LIN {X 0,Y 467.549,Z 626.363,A -85,B 0,C 180,E1 -7509.148,E2 -7509.148} C_VEL
LIN {X 0,Y 467.561,Z 626.367,A -85,B 0,C 180,E1 -7511.405,E2 -7511.405} C_VEL
LIN {X 0,Y 467.569,Z 626.37,A -85,B 0,C 180,E1 -7515.052,E2 -7515.052} C_VEL
LIN {X 0,Y 467.563,Z 626.367,A -85,B 0,C 180,E1 -7518.726,E2 -7518.726} C_VEL
LIN {X 0,Y 467.552,Z 626.355,A -85,B 0,C 180,E1 -7521.954,E2 -7521.954} C_VEL
LIN {X 0,Y 467.559,Z 626.366,A -85,B 0,C 180,E1 -7525.166,E2 -7525.166} C_VEL
LIN {X 0,Y 467.585,Z 626.36,A -85,B 0,C 180,E1 -7528.26,E2 -7528.26} C_VEL
LIN {X 0,Y 467.556,Z 626.368,A -85,B 0,C 180,E1 -7531.249,E2 -7531.249} C_VEL
LIN {X 0,Y 467.579,Z 626.36,A -85,B 0,C 180,E1 -7534.401,E2 -7534.401} C_VEL
LIN {X 0,Y 467.579,Z 626.359,A -85,B 0,C 180,E1 -7536.996,E2 -7536.996} C_VEL
LIN {X 0,Y 467.626,Z 626.359,A -85,B 0,C 180,E1 -7539.777,E2 -7539.777} C_VEL
LIN {X 0,Y 467.601,Z 626.35,A -85,B 0,C 180,E1 -7542.506,E2 -7542.506} C_VEL
LIN {X 0,Y 467.609,Z 626.36,A -85,B 0,C 180,E1 -7545.196,E2 -7545.196} C_VEL
LIN {X 0,Y 467.659,Z 626.352,A -85,B 0,C 180,E1 -7547.854,E2 -7547.854} C_VEL
LIN {X 0,Y 467.673,Z 626.349,A -85,B 0,C 180,E1 -7551.357,E2 -7551.357} C_VEL
LIN {X 0,Y 467.716,Z 626.348,A -85,B 0,C 180,E1 -7553.962,E2 -7553.962} C_VEL
LIN {X 0,Y 467.854,Z 626.329,A -85,B 0,C 180,E1 -7557.417,E2 -7557.417} C_VEL
LIN {X 0,Y 467.885,Z 626.326,A -85,B 0,C 180,E1 -7560,E2 -7560} C_VEL
LIN {X 0,Y 467.861,Z 626.327,A -85,B 0,C 180,E1 -7562.583,E2 -7562.583} C_VEL
LIN {X 0,Y 467.725,Z 626.348,A -85,B 0,C 180,E1 -7566.037,E2 -7566.037} C_VEL
LIN {X 0,Y 467.683,Z 626.349,A -85,B 0,C 180,E1 -7568.643,E2 -7568.643} C_VEL
LIN {X 0,Y 467.659,Z 626.358,A -85,B 0,C 180,E1 -7572.145,E2 -7572.145} C_VEL
LIN {X 0,Y 467.67,Z 626.353,A -85,B 0,C 180,E1 -7575.893,E2 -7575.893} C_VEL
LIN {X 0,Y 467.627,Z 626.353,A -85,B 0,C 180,E1 -7579.307,E2 -7579.307} C_VEL
LIN {X 0,Y 467.537,Z 626.373,A -85,B 0,C 180,E1 -7582.074,E2 -7582.074} C_VEL
LIN {X 0,Y 467.588,Z 626.361,A -85,B 0,C 180,E1 -7584.888,E2 -7584.888} C_VEL
LIN {X 0,Y 467.622,Z 626.356,A -85,B 0,C 180,E1 -7587.769,E2 -7587.769} C_VEL
LIN {X 0,Y 467.57,Z 626.362,A -85,B 0,C 180,E1 -7591.045,E2 -7591.045} C_VEL
LIN {X 0,Y 467.59,Z 626.366,A -85,B 0,C 180,E1 -7594.242,E2 -7594.242} C_VEL
LIN {X 0,Y 467.55,Z 626.366,A -85,B 0,C 180,E1 -7597.186,E2 -7597.186} C_VEL
LIN {X 0,Y 467.597,Z 626.364,A -85,B 0,C 180,E1 -7600.262,E2 -7600.262} C_VEL
LIN {X 0,Y 467.588,Z 626.368,A -85,B 0,C 180,E1 -7602.567,E2 -7602.567} C_VEL
LIN {X 0,Y 467.572,Z 626.364,A -85,B 0,C 180,E1 -7605.053,E2 -7605.053} C_VEL
LIN {X 0,Y 467.59,Z 626.36,A -85,B 0,C 180,E1 -7607.44,E2 -7607.44} C_VEL
LIN {X 0,Y 467.584,Z 626.368,A -85,B 0,C 180,E1 -7610.855,E2 -7610.855} C_VEL
LIN {X 0,Y 467.565,Z 626.368,A -85,B 0,C 180,E1 -7614.26,E2 -7614.26} C_VEL
LIN {X 0,Y 467.584,Z 626.365,A -85,B 0,C 180,E1 -7617.321,E2 -7617.321} C_VEL
LIN {X 0,Y 467.572,Z 626.369,A -85,B 0,C 180,E1 -7620.667,E2 -7620.667} C_VEL
LIN {X 0,Y 467.653,Z 626.484,A -85,B 0,C 180,E1 -7621.654,E2 -7621.654} C_VEL
LIN {X 0,Y 470.749,Z 640.596,A -85,B 0,C 180,E1 -7624.125,E2 -7624.125} C_VEL
LIN {X 0,Y 471.136,Z 644.928,A -85,B 0,C 180,E1 -7624.84,E2 -7624.84} C_VEL
LIN {X 0,Y 469.974,Z 666.892,A -85,B 0,C 180,E1 -7628.277,E2 -7628.277} C_VEL
LIN {X 0,Y 469.639,Z 674.02,A -85,B 0,C 180,E1 -7629.383,E2 -7629.383} C_VEL
LIN {X 0,Y 473.403,Z 695.857,A -85,B 0,C 180,E1 -7629.896,E2 -7629.896} C_VEL
LIN {X 0,Y 472.198,Z 812.498,A -85,B 0,C 180,E1 -7631.702,E2 -7631.702} C_VEL
LIN {X 0,Y 471.755,Z 827.182,A -85,B 0,C 180,E1 -7632.108,E2 -7632.108} C_VEL
LIN {X 0,Y 471.281,Z 840.517,A -85,B 0,C 180,E1 -7632.647,E2 -7632.647} C_VEL
LIN {X 0,Y 470.687,Z 853.287,A -85,B 0,C 180,E1 -7633.329,E2 -7633.329} C_VEL
LIN {X 0,Y 470.047,Z 865.621,A -85,B 0,C 180,E1 -7634.165,E2 -7634.165} C_VEL
LIN {X 0,Y 469.361,Z 877.324,A -85,B 0,C 180,E1 -7635.142,E2 -7635.142} C_VEL
LIN {X 0,Y 468.755,Z 887.065,A -85,B 0,C 180,E1 -7636.12,E2 -7636.12} C_VEL
LIN {X 0,Y 468.168,Z 897.352,A -85,B 0,C 180,E1 -7637.359,E2 -7637.359} C_VEL
LIN {X 0,Y 467.713,Z 906.781,A -85,B 0,C 180,E1 -7638.735,E2 -7638.735} C_VEL
LIN {X 0,Y 467.263,Z 915.33,A -85,B 0,C 180,E1 -7640.258,E2 -7640.258} C_VEL
LIN {X 0,Y 466.964,Z 922.224,A -85,B 0,C 180,E1 -7641.78,E2 -7641.78} C_VEL
LIN {X 0,Y 466.825,Z 926.979,A -85,B 0,C 180,E1 -7643.082,E2 -7643.082} C_VEL
LIN {X 0,Y 466.757,Z 931.907,A -85,B 0,C 180,E1 -7644.817,E2 -7644.817} C_VEL
LIN {X 0,Y 466.681,Z 935.332,A -85,B 0,C 180,E1 -7646.546,E2 -7646.546} C_VEL
LIN {X 0,Y 466.625,Z 937.357,A -85,B 0,C 180,E1 -7648.274,E2 -7648.274} C_VEL
LIN {X 0,Y 466.596,Z 938.027,A -85,B 0,C 180,E1 -7650,E2 -7650} C_VEL
LIN {X 0,Y 466.625,Z 937.354,A -85,B 0,C 180,E1 -7651.726,E2 -7651.726} C_VEL
LIN {X 0,Y 466.681,Z 935.327,A -85,B 0,C 180,E1 -7653.453,E2 -7653.453} C_VEL
LIN {X 0,Y 466.757,Z 931.896,A -85,B 0,C 180,E1 -7655.183,E2 -7655.183} C_VEL
LIN {X 0,Y 466.822,Z 926.957,A -85,B 0,C 180,E1 -7656.917,E2 -7656.917} C_VEL
LIN {X 0,Y 467.051,Z 920.373,A -85,B 0,C 180,E1 -7658.654,E2 -7658.654} C_VEL
LIN {X 0,Y 467.334,Z 913.049,A -85,B 0,C 180,E1 -7660.178,E2 -7660.178} C_VEL
LIN {X 0,Y 467.853,Z 903.988,A -85,B 0,C 180,E1 -7661.7,E2 -7661.7} C_VEL
LIN {X 0,Y 468.348,Z 894.482,A -85,B 0,C 180,E1 -7663.008,E2 -7663.008} C_VEL
LIN {X 0,Y 468.929,Z 883.967,A -85,B 0,C 180,E1 -7664.206,E2 -7664.206} C_VEL
LIN {X 0,Y 469.577,Z 872.377,A -85,B 0,C 180,E1 -7665.295,E2 -7665.295} C_VEL
LIN {X 0,Y 470.364,Z 859.535,A -85,B 0,C 180,E1 -7666.269,E2 -7666.269} C_VEL
LIN {X 0,Y 470.997,Z 847.029,A -85,B 0,C 180,E1 -7667.027,E2 -7667.027} C_VEL
LIN {X 0,Y 471.554,Z 833.87,A -85,B 0,C 180,E1 -7667.644,E2 -7667.644} C_VEL
LIN {X 0,Y 472.024,Z 819.661,A -85,B 0,C 180,E1 -7668.128,E2 -7668.128} C_VEL
LIN {X 0,Y 472.336,Z 805.526,A -85,B 0,C 180,E1 -7668.432,E2 -7668.432} C_VEL
LIN {X 0,Y 473.472,Z 695.812,A -85,B 0,C 180,E1 -7670.118,E2 -7670.118} C_VEL
LIN {X 0,Y 469.655,Z 673.893,A -85,B 0,C 180,E1 -7670.657,E2 -7670.657} C_VEL
LIN {X 0,Y 470.482,Z 656.971,A -85,B 0,C 180,E1 -7673.319,E2 -7673.319} C_VEL
LIN {X 0,Y 471.209,Z 643.957,A -85,B 0,C 180,E1 -7675.391,E2 -7675.391} C_VEL
LIN {X 0,Y 469.983,Z 636.708,A -85,B 0,C 180,E1 -7676.655,E2 -7676.655} C_VEL
LIN {X 0,Y 467.61,Z 626.365,A -85,B 0,C 180,E1 -7678.563,E2 -7678.563} C_VEL
LIN {X 0,Y 467.585,Z 626.363,A -85,B 0,C 180,E1 -7681.74,E2 -7681.74} C_VEL
LIN {X 0,Y 467.57,Z 626.364,A -85,B 0,C 180,E1 -7684.832,E2 -7684.832} C_VEL
LIN {X 0,Y 467.568,Z 626.364,A -85,B 0,C 180,E1 -7688.044,E2 -7688.044} C_VEL
LIN {X 0,Y 467.583,Z 626.364,A -85,B 0,C 180,E1 -7691.277,E2 -7691.277} C_VEL
LIN {X 0,Y 467.567,Z 626.363,A -85,B 0,C 180,E1 -7693.823,E2 -7693.823} C_VEL
LIN {X 0,Y 467.557,Z 626.365,A -85,B 0,C 180,E1 -7696.256,E2 -7696.256} C_VEL
LIN {X 0,Y 467.585,Z 626.358,A -85,B 0,C 180,E1 -7698.722,E2 -7698.722} C_VEL
LIN {X 0,Y 467.576,Z 626.367,A -85,B 0,C 180,E1 -7701.407,E2 -7701.407} C_VEL
LIN {X 0,Y 467.564,Z 626.365,A -85,B 0,C 180,E1 -7704.26,E2 -7704.26} C_VEL
LIN {X 0,Y 467.583,Z 626.363,A -85,B 0,C 180,E1 -7707.321,E2 -7707.321} C_VEL
LIN {X 0,Y 467.571,Z 626.361,A -85,B 0,C 180,E1 -7710.667,E2 -7710.667} C_VEL
LIN {X 0,Y 467.618,Z 626.357,A -85,B 0,C 180,E1 -7713.2,E2 -7713.2} C_VEL
LIN {X 0,Y 467.594,Z 626.359,A -85,B 0,C 180,E1 -7716.468,E2 -7716.468} C_VEL
LIN {X 0,Y 467.626,Z 626.362,A -85,B 0,C 180,E1 -7719.777,E2 -7719.777} C_VEL
LIN {X 0,Y 467.611,Z 626.359,A -85,B 0,C 180,E1 -7722.507,E2 -7722.507} C_VEL
LIN {X 0,Y 467.608,Z 626.358,A -85,B 0,C 180,E1 -7725.197,E2 -7725.197} C_VEL
LIN {X 0,Y 467.658,Z 626.355,A -85,B 0,C 180,E1 -7727.855,E2 -7727.855} C_VEL
LIN {X 0,Y 467.683,Z 626.345,A -85,B 0,C 180,E1 -7731.357,E2 -7731.357} C_VEL
LIN {X 0,Y 467.739,Z 626.347,A -85,B 0,C 180,E1 -7733.963,E2 -7733.963} C_VEL
LIN {X 0,Y 467.861,Z 626.326,A -85,B 0,C 180,E1 -7737.417,E2 -7737.417} C_VEL
LIN {X 0,Y 467.884,Z 626.327,A -85,B 0,C 180,E1 -7740,E2 -7740} C_VEL
LIN {X 0,Y 467.861,Z 626.333,A -85,B 0,C 180,E1 -7742.583,E2 -7742.583} C_VEL
LIN {X 0,Y 467.737,Z 626.34,A -85,B 0,C 180,E1 -7746.038,E2 -7746.038} C_VEL
LIN {X 0,Y 467.682,Z 626.354,A -85,B 0,C 180,E1 -7748.643,E2 -7748.643} C_VEL
LIN {X 0,Y 467.658,Z 626.354,A -85,B 0,C 180,E1 -7752.146,E2 -7752.146} C_VEL
LIN {X 0,Y 467.641,Z 626.351,A -85,B 0,C 180,E1 -7755.695,E2 -7755.695} C_VEL
LIN {X 0,Y 467.615,Z 626.36,A -85,B 0,C 180,E1 -7758.763,E2 -7758.763} C_VEL
LIN {X 0,Y 467.583,Z 626.364,A -85,B 0,C 180,E1 -7761.268,E2 -7761.268} C_VEL
LIN {X 0,Y 467.571,Z 626.36,A -85,B 0,C 180,E1 -7763.944,E2 -7763.944} C_VEL
LIN {X 0,Y 467.569,Z 626.367,A -85,B 0,C 180,E1 -7766.804,E2 -7766.804} C_VEL
LIN {X 0,Y 467.549,Z 626.357,A -85,B 0,C 180,E1 -7769.739,E2 -7769.739} C_VEL
LIN {X 0,Y 467.582,Z 626.368,A -85,B 0,C 180,E1 -7772.759,E2 -7772.759} C_VEL
LIN {X 0,Y 467.555,Z 626.365,A -85,B 0,C 180,E1 -7775.89,E2 -7775.89} C_VEL
LIN {X 0,Y 467.555,Z 626.369,A -85,B 0,C 180,E1 -7779.148,E2 -7779.148} C_VEL
LIN {X 0,Y 467.565,Z 626.364,A -85,B 0,C 180,E1 -7781.405,E2 -7781.405} C_VEL
LIN {X 0,Y 467.568,Z 626.366,A -85,B 0,C 180,E1 -7785.053,E2 -7785.053} C_VEL
LIN {X 0,Y 467.563,Z 626.368,A -85,B 0,C 180,E1 -7788.726,E2 -7788.726} C_VEL
LIN {X 0,Y 467.566,Z 626.367,A -85,B 0,C 180,E1 -7791.956,E2 -7791.956} C_VEL
LIN {X 0,Y 467.56,Z 626.369,A -85,B 0,C 180,E1 -7795.167,E2 -7795.167} C_VEL
LIN {X 0,Y 467.579,Z 626.366,A -85,B 0,C 180,E1 -7798.26,E2 -7798.26} C_VEL
LIN {X 0,Y 467.617,Z 626.495,A -85,B 0,C 180,E1 -7801.315,E2 -7801.315} C_VEL
LIN {X 0,Y 469.754,Z 637.568,A -85,B 0,C 180,E1 -7803.66,E2 -7803.66} C_VEL
LIN {X 0,Y 469.686,Z 641.571,A -85,B 0,C 180,E1 -7804.419,E2 -7804.419} C_VEL
LIN {X 0,Y 473.504,Z 658.762,A -85,B 0,C 180,E1 -7804.878,E2 -7804.878} C_VEL
LIN {X 0,Y 473.154,Z 702.769,A -85,B 0,C 180,E1 -7805.562,E2 -7805.562} C_VEL
LIN {X 0,Y 472.453,Z 708.622,A -85,B 0,C 180,E1 -7805.623,E2 -7805.623} C_VEL
LIN {X 0,Y 466.856,Z 727.666,A -85,B 0,C 180,E1 -7805.673,E2 -7805.673} C_VEL
LIN {X 0,Y 466.209,Z 733.515,A -85,B 0,C 180,E1 -7805.738,E2 -7805.738} C_VEL
LIN {X 0,Y 465.795,Z 778.177,A -85,B 0,C 180,E1 -7806.462,E2 -7806.462} C_VEL
LIN {X 0,Y 465.39,Z 792.175,A -85,B 0,C 180,E1 -7806.852,E2 -7806.852} C_VEL
LIN {X 0,Y 464.798,Z 805.625,A -85,B 0,C 180,E1 -7807.396,E2 -7807.396} C_VEL
LIN {X 0,Y 464.197,Z 818.732,A -85,B 0,C 180,E1 -7808.11,E2 -7808.11} C_VEL
LIN {X 0,Y 463.49,Z 831.624,A -85,B 0,C 180,E1 -7809.008,E2 -7809.008} C_VEL
LIN {X 0,Y 462.779,Z 843.773,A -85,B 0,C 180,E1 -7810.066,E2 -7810.066} C_VEL
LIN {X 0,Y 462.135,Z 853.964,A -85,B 0,C 180,E1 -7811.146,E2 -7811.146} C_VEL
LIN {X 0,Y 461.43,Z 864.506,A -85,B 0,C 180,E1 -7812.494,E2 -7812.494} C_VEL
LIN {X 0,Y 460.921,Z 873.302,A -85,B 0,C 180,E1 -7813.866,E2 -7813.866} C_VEL
LIN {X 0,Y 460.384,Z 881.398,A -85,B 0,C 180,E1 -7815.411,E2 -7815.411} C_VEL
LIN {X 0,Y 460.086,Z 887.146,A -85,B 0,C 180,E1 -7816.754,E2 -7816.754} C_VEL
LIN {X 0,Y 459.861,Z 891.486,A -85,B 0,C 180,E1 -7817.99,E2 -7817.99} C_VEL
LIN {X 0,Y 459.735,Z 895.569,A -85,B 0,C 180,E1 -7819.43,E2 -7819.43} C_VEL
LIN {X 0,Y 459.588,Z 899.217,A -85,B 0,C 180,E1 -7821.204,E2 -7821.204} C_VEL
LIN {X 0,Y 459.612,Z 901.449,A -85,B 0,C 180,E1 -7822.974,E2 -7822.974} C_VEL
LIN {X 0,Y 459.573,Z 902.34,A -85,B 0,C 180,E1 -7824.736,E2 -7824.736} C_VEL
LIN {X 0,Y 459.586,Z 901.914,A -85,B 0,C 180,E1 -7826.493,E2 -7826.493} C_VEL
LIN {X 0,Y 459.595,Z 900.176,A -85,B 0,C 180,E1 -7828.248,E2 -7828.248} C_VEL
LIN {X 0,Y 459.562,Z 897.101,A -85,B 0,C 180,E1 -7830,E2 -7830} C_VEL
LIN {X 0,Y 459.699,Z 892.579,A -85,B 0,C 180,E1 -7831.752,E2 -7831.752} C_VEL
LIN {X 0,Y 460.114,Z 886.426,A -85,B 0,C 180,E1 -7833.503,E2 -7833.503} C_VEL
LIN {X 0,Y 460.536,Z 879.59,A -85,B 0,C 180,E1 -7835.034,E2 -7835.034} C_VEL
LIN {X 0,Y 461.037,Z 871.138,A -85,B 0,C 180,E1 -7836.565,E2 -7836.565} C_VEL
LIN {X 0,Y 461.445,Z 862.335,A -85,B 0,C 180,E1 -7837.879,E2 -7837.879} C_VEL
LIN {X 0,Y 462.271,Z 851.65,A -85,B 0,C 180,E1 -7839.186,E2 -7839.186} C_VEL
LIN {X 0,Y 462.963,Z 840.842,A -85,B 0,C 180,E1 -7840.275,E2 -7840.275} C_VEL
LIN {X 0,Y 463.629,Z 829.013,A -85,B 0,C 180,E1 -7841.255,E2 -7841.255} C_VEL
LIN {X 0,Y 464.374,Z 815.847,A -85,B 0,C 180,E1 -7842.122,E2 -7842.122} C_VEL
LIN {X 0,Y 464.924,Z 803.168,A -85,B 0,C 180,E1 -7842.772,E2 -7842.772} C_VEL
LIN {X 0,Y 465.319,Z 789.688,A -85,B 0,C 180,E1 -7843.289,E2 -7843.289} C_VEL
LIN {X 0,Y 465.578,Z 776.034,A -85,B 0,C 180,E1 -7843.643,E2 -7843.643} C_VEL
LIN {X 0,Y 466.828,Z 659.89,A -85,B 0,C 180,E1 -7845.459,E2 -7845.459} C_VEL
LIN {X 0,Y 462.732,Z 641.579,A -85,B 0,C 180,E1 -7845.949,E2 -7845.949} C_VEL
LIN {X 0,Y 462.545,Z 637.217,A -85,B 0,C 180,E1 -7846.815,E2 -7846.815} C_VEL
LIN {X 0,Y 460.573,Z 627.244,A -85,B 0,C 180,E1 -7848.939,E2 -7848.939} C_VEL
LIN {X 0,Y 460.52,Z 627.246,A -85,B 0,C 180,E1 -7851.486,E2 -7851.486} C_VEL
LIN {X 0,Y 460.516,Z 627.248,A -85,B 0,C 180,E1 -7854.334,E2 -7854.334} C_VEL
LIN {X 0,Y 460.488,Z 627.25,A -85,B 0,C 180,E1 -7857.249,E2 -7857.249} C_VEL
LIN {X 0,Y 460.496,Z 627.248,A -85,B 0,C 180,E1 -7860.241,E2 -7860.241} C_VEL
LIN {X 0,Y 460.504,Z 627.247,A -85,B 0,C 180,E1 -7863.327,E2 -7863.327} C_VEL
LIN {X 0,Y 460.463,Z 627.252,A -85,B 0,C 180,E1 -7866.531,E2 -7866.531} C_VEL
LIN {X 0,Y 460.513,Z 627.234,A -85,B 0,C 180,E1 -7869.865,E2 -7869.865} C_VEL
LIN {X 0,Y 460.465,Z 627.255,A -85,B 0,C 180,E1 -7872.893,E2 -7872.893} C_VEL
LIN {X 0,Y 460.506,Z 627.243,A -85,B 0,C 180,E1 -7875.831,E2 -7875.831} C_VEL
LIN {X 0,Y 460.517,Z 627.248,A -85,B 0,C 180,E1 -7878.987,E2 -7878.987} C_VEL
LIN {X 0,Y 460.495,Z 627.234,A -85,B 0,C 180,E1 -7882.376,E2 -7882.376} C_VEL
LIN {X 0,Y 460.539,Z 627.242,A -85,B 0,C 180,E1 -7885.623,E2 -7885.623} C_VEL
LIN {X 0,Y 460.541,Z 627.239,A -85,B 0,C 180,E1 -7888.744,E2 -7888.744} C_VEL
LIN {X 0,Y 460.521,Z 627.244,A -85,B 0,C 180,E1 -7891.765,E2 -7891.765} C_VEL
LIN {X 0,Y 460.523,Z 627.24,A -85,B 0,C 180,E1 -7894.703,E2 -7894.703} C_VEL
LIN {X 0,Y 460.514,Z 627.248,A -85,B 0,C 180,E1 -7897.571,E2 -7897.571} C_VEL
LIN {X 0,Y 460.571,Z 627.233,A -85,B 0,C 180,E1 -7900.384,E2 -7900.384} C_VEL
LIN {X 0,Y 460.608,Z 627.23,A -85,B 0,C 180,E1 -7904.059,E2 -7904.059} C_VEL
LIN {X 0,Y 460.612,Z 627.232,A -85,B 0,C 180,E1 -7907.666,E2 -7907.666} C_VEL
LIN {X 0,Y 460.623,Z 627.226,A -85,B 0,C 180,E1 -7911.223,E2 -7911.223} C_VEL
LIN {X 0,Y 460.68,Z 627.226,A -85,B 0,C 180,E1 -7913.869,E2 -7913.869} C_VEL
LIN {X 0,Y 460.795,Z 627.208,A -85,B 0,C 180,E1 -7917.377,E2 -7917.377} C_VEL
LIN {X 0,Y 460.855,Z 627.201,A -85,B 0,C 180,E1 -7920,E2 -7920} C_VEL
LIN {X 0,Y 460.802,Z 627.206,A -85,B 0,C 180,E1 -7922.622,E2 -7922.622} C_VEL
LIN {X 0,Y 460.689,Z 627.224,A -85,B 0,C 180,E1 -7926.13,E2 -7926.13} C_VEL
LIN {X 0,Y 460.63,Z 627.228,A -85,B 0,C 180,E1 -7928.776,E2 -7928.776} C_VEL
LIN {X 0,Y 460.616,Z 627.232,A -85,B 0,C 180,E1 -7932.445,E2 -7932.445} C_VEL
LIN {X 0,Y 460.625,Z 627.231,A -85,B 0,C 180,E1 -7936.007,E2 -7936.007} C_VEL
LIN {X 0,Y 460.572,Z 627.234,A -85,B 0,C 180,E1 -7939.615,E2 -7939.615} C_VEL
LIN {X 0,Y 460.513,Z 627.244,A -85,B 0,C 180,E1 -7942.428,E2 -7942.428} C_VEL
LIN {X 0,Y 460.555,Z 627.239,A -85,B 0,C 180,E1 -7945.798,E2 -7945.798} C_VEL
LIN {X 0,Y 460.554,Z 627.241,A -85,B 0,C 180,E1 -7948.233,E2 -7948.233} C_VEL
LIN {X 0,Y 460.523,Z 627.24,A -85,B 0,C 180,E1 -7951.283,E2 -7951.283} C_VEL
LIN {X 0,Y 460.534,Z 627.246,A -85,B 0,C 180,E1 -7954.505,E2 -7954.505} C_VEL
LIN {X 0,Y 460.531,Z 627.24,A -85,B 0,C 180,E1 -7957.62,E2 -7957.62} C_VEL
LIN {X 0,Y 460.56,Z 627.241,A -85,B 0,C 180,E1 -7960.272,E2 -7960.272} C_VEL
LIN {X 0,Y 460.501,Z 627.243,A -85,B 0,C 180,E1 -7963.375,E2 -7963.375} C_VEL
LIN {X 0,Y 460.51,Z 627.244,A -85,B 0,C 180,E1 -7966.626,E2 -7966.626} C_VEL
LIN {X 0,Y 460.544,Z 627.239,A -85,B 0,C 180,E1 -7969.73,E2 -7969.73} C_VEL
LIN {X 0,Y 460.529,Z 627.247,A -85,B 0,C 180,E1 -7972.519,E2 -7972.519} C_VEL
LIN {X 0,Y 460.55,Z 627.24,A -85,B 0,C 180,E1 -7975.624,E2 -7975.624} C_VEL
LIN {X 0,Y 460.538,Z 627.239,A -85,B 0,C 180,E1 -7978.744,E2 -7978.744} C_VEL
LIN {X 0,Y 460.58,Z 627.369,A -85,B 0,C 180,E1 -7981.396,E2 -7981.396} C_VEL
LIN {X 0,Y 463.744,Z 641.575,A -85,B 0,C 180,E1 -7983.928,E2 -7983.928} C_VEL
LIN {X 0,Y 464.25,Z 646.024,A -85,B 0,C 180,E1 -7984.681,E2 -7984.681} C_VEL
LIN {X 0,Y 463.023,Z 668.116,A -85,B 0,C 180,E1 -7988.19,E2 -7988.19} C_VEL
LIN {X 0,Y 462.729,Z 673.729,A -85,B 0,C 180,E1 -7989.073,E2 -7989.073} C_VEL
LIN {X 0,Y 466.702,Z 697.353,A -85,B 0,C 180,E1 -7989.634,E2 -7989.634} C_VEL
LIN {X 0,Y 465.446,Z 811.857,A -85,B 0,C 180,E1 -7991.427,E2 -7991.427} C_VEL
LIN {X 0,Y 464.988,Z 826.608,A -85,B 0,C 180,E1 -7991.836,E2 -7991.836} C_VEL
LIN {X 0,Y 464.433,Z 840.997,A -85,B 0,C 180,E1 -7992.429,E2 -7992.429} C_VEL
LIN {X 0,Y 463.771,Z 854.532,A -85,B 0,C 180,E1 -7993.178,E2 -7993.178} C_VEL
LIN {X 0,Y 463.086,Z 866.71,A -85,B 0,C 180,E1 -7994.034,E2 -7994.034} C_VEL
LIN {X 0,Y 462.379,Z 878.185,A -85,B 0,C 180,E1 -7995.025,E2 -7995.025} C_VEL
LIN {X 0,Y 461.69,Z 888.726,A -85,B 0,C 180,E1 -7996.128,E2 -7996.128} C_VEL
LIN {X 0,Y 461.104,Z 899.133,A -85,B 0,C 180,E1 -7997.444,E2 -7997.444} C_VEL
LIN {X 0,Y 460.605,Z 907.865,A -85,B 0,C 180,E1 -7998.782,E2 -7998.782} C_VEL
LIN {X 0,Y 460.181,Z 916.152,A -85,B 0,C 180,E1 -8000.329,E2 -8000.329} C_VEL
LIN {X 0,Y 459.911,Z 921.951,A -85,B 0,C 180,E1 -8001.653,E2 -8001.653} C_VEL
LIN {X 0,Y 459.734,Z 926.705,A -85,B 0,C 180,E1 -8002.975,E2 -8002.975} C_VEL
LIN {X 0,Y 459.667,Z 931.634,A -85,B 0,C 180,E1 -8004.736,E2 -8004.736} C_VEL
LIN {X 0,Y 459.577,Z 935.059,A -85,B 0,C 180,E1 -8006.493,E2 -8006.493} C_VEL
LIN {X 0,Y 459.535,Z 937.085,A -85,B 0,C 180,E1 -8008.247,E2 -8008.247} C_VEL
LIN {X 0,Y 459.528,Z 937.755,A -85,B 0,C 180,E1 -8010,E2 -8010} C_VEL
LIN {X 0,Y 459.535,Z 937.081,A -85,B 0,C 180,E1 -8011.753,E2 -8011.753} C_VEL
LIN {X 0,Y 459.577,Z 935.052,A -85,B 0,C 180,E1 -8013.507,E2 -8013.507} C_VEL
LIN {X 0,Y 459.667,Z 931.62,A -85,B 0,C 180,E1 -8015.263,E2 -8015.263} C_VEL
LIN {X 0,Y 459.733,Z 926.68,A -85,B 0,C 180,E1 -8017.025,E2 -8017.025} C_VEL
LIN {X 0,Y 459.982,Z 920.094,A -85,B 0,C 180,E1 -8018.789,E2 -8018.789} C_VEL
LIN {X 0,Y 460.301,Z 912.773,A -85,B 0,C 180,E1 -8020.335,E2 -8020.335} C_VEL
LIN {X 0,Y 460.827,Z 903.717,A -85,B 0,C 180,E1 -8021.881,E2 -8021.881} C_VEL
LIN {X 0,Y 461.36,Z 894.226,A -85,B 0,C 180,E1 -8023.209,E2 -8023.209} C_VEL
LIN {X 0,Y 462.02,Z 883.731,A -85,B 0,C 180,E1 -8024.423,E2 -8024.423} C_VEL
LIN {X 0,Y 462.695,Z 872.17,A -85,B 0,C 180,E1 -8025.528,E2 -8025.528} C_VEL
LIN {X 0,Y 463.501,Z 859.362,A -85,B 0,C 180,E1 -8026.517,E2 -8026.517} C_VEL
LIN {X 0,Y 464.223,Z 846.549,A -85,B 0,C 180,E1 -8027.303,E2 -8027.303} C_VEL
LIN {X 0,Y 464.829,Z 833.021,A -85,B 0,C 180,E1 -8027.942,E2 -8027.942} C_VEL
LIN {X 0,Y 465.358,Z 818.507,A -85,B 0,C 180,E1 -8028.434,E2 -8028.434} C_VEL
LIN {X 0,Y 465.659,Z 804.149,A -85,B 0,C 180,E1 -8028.735,E2 -8028.735} C_VEL
LIN {X 0,Y 466.701,Z 695.75,A -85,B 0,C 180,E1 -8030.432,E2 -8030.432} C_VEL
LIN {X 0,Y 462.804,Z 673.619,A -85,B 0,C 180,E1 -8030.991,E2 -8030.991} C_VEL
LIN {X 0,Y 463.901,Z 653.933,A -85,B 0,C 180,E1 -8034.145,E2 -8034.145} C_VEL
LIN {X 0,Y 464.354,Z 645.272,A -85,B 0,C 180,E1 -8035.553,E2 -8035.553} C_VEL
LIN {X 0,Y 462.453,Z 635.305,A -85,B 0,C 180,E1 -8037.339,E2 -8037.339} C_VEL
LIN {X 0,Y 460.565,Z 627.243,A -85,B 0,C 180,E1 -8038.854,E2 -8038.854} C_VEL
LIN {X 0,Y 460.533,Z 627.239,A -85,B 0,C 180,E1 -8042.284,E2 -8042.284} C_VEL
LIN {X 0,Y 460.515,Z 627.242,A -85,B 0,C 180,E1 -8045.445,E2 -8045.445} C_VEL
LIN {X 0,Y 460.552,Z 627.24,A -85,B 0,C 180,E1 -8048.899,E2 -8048.899} C_VEL
LIN {X 0,Y 460.524,Z 627.243,A -85,B 0,C 180,E1 -8052.181,E2 -8052.181} C_VEL
LIN {X 0,Y 460.518,Z 627.246,A -85,B 0,C 180,E1 -8055.412,E2 -8055.412} C_VEL
LIN {X 0,Y 460.536,Z 627.236,A -85,B 0,C 180,E1 -8058.397,E2 -8058.397} C_VEL
LIN {X 0,Y 460.545,Z 627.242,A -85,B 0,C 180,E1 -8061.269,E2 -8061.269} C_VEL
LIN {X 0,Y 460.515,Z 627.242,A -85,B 0,C 180,E1 -8064.555,E2 -8064.555} C_VEL
LIN {X 0,Y 460.533,Z 627.234,A -85,B 0,C 180,E1 -8067.716,E2 -8067.716} C_VEL
LIN {X 0,Y 460.541,Z 627.236,A -85,B 0,C 180,E1 -8070.769,E2 -8070.769} C_VEL
LIN {X 0,Y 460.564,Z 627.238,A -85,B 0,C 180,E1 -8073.735,E2 -8073.735} C_VEL
LIN {X 0,Y 460.548,Z 627.236,A -85,B 0,C 180,E1 -8076.624,E2 -8076.624} C_VEL
LIN {X 0,Y 460.554,Z 627.239,A -85,B 0,C 180,E1 -8079.453,E2 -8079.453} C_VEL
LIN {X 0,Y 460.562,Z 627.24,A -85,B 0,C 180,E1 -8082.23,E2 -8082.23} C_VEL
LIN {X 0,Y 460.571,Z 627.234,A -85,B 0,C 180,E1 -8084.965,E2 -8084.965} C_VEL
LIN {X 0,Y 460.613,Z 627.232,A -85,B 0,C 180,E1 -8088.56,E2 -8088.56} C_VEL
LIN {X 0,Y 460.697,Z 627.222,A -85,B 0,C 180,E1 -8092.109,E2 -8092.109} C_VEL
LIN {X 0,Y 460.698,Z 627.217,A -85,B 0,C 180,E1 -8094.749,E2 -8094.749} C_VEL
LIN {X 0,Y 460.802,Z 627.206,A -85,B 0,C 180,E1 -8097.378,E2 -8097.378} C_VEL
LIN {X 0,Y 460.854,Z 627.203,A -85,B 0,C 180,E1 -8100,E2 -8100} C_VEL
LIN {X 0,Y 460.802,Z 627.212,A -85,B 0,C 180,E1 -8102.623,E2 -8102.623} C_VEL
LIN {X 0,Y 460.703,Z 627.217,A -85,B 0,C 180,E1 -8106.13,E2 -8106.13} C_VEL
LIN {X 0,Y 460.629,Z 627.23,A -85,B 0,C 180,E1 -8108.776,E2 -8108.776} C_VEL
LIN {X 0,Y 460.616,Z 627.235,A -85,B 0,C 180,E1 -8112.445,E2 -8112.445} C_VEL
LIN {X 0,Y 460.602,Z 627.229,A -85,B 0,C 180,E1 -8115.998,E2 -8115.998} C_VEL
LIN {X 0,Y 460.57,Z 627.231,A -85,B 0,C 180,E1 -8119.616,E2 -8119.616} C_VEL
LIN {X 0,Y 460.513,Z 627.247,A -85,B 0,C 180,E1 -8122.429,E2 -8122.429} C_VEL
LIN {X 0,Y 460.552,Z 627.238,A -85,B 0,C 180,E1 -8125.797,E2 -8125.797} C_VEL
LIN {X 0,Y 460.529,Z 627.235,A -85,B 0,C 180,E1 -8128.235,E2 -8128.235} C_VEL
LIN {X 0,Y 460.523,Z 627.245,A -85,B 0,C 180,E1 -8131.283,E2 -8131.283} C_VEL
LIN {X 0,Y 460.525,Z 627.241,A -85,B 0,C 180,E1 -8134.504,E2 -8134.504} C_VEL
LIN {X 0,Y 460.503,Z 627.246,A -85,B 0,C 180,E1 -8137.623,E2 -8137.623} C_VEL
LIN {X 0,Y 460.526,Z 627.237,A -85,B 0,C 180,E1 -8140.267,E2 -8140.267} C_VEL
LIN {X 0,Y 460.505,Z 627.25,A -85,B 0,C 180,E1 -8143.375,E2 -8143.375} C_VEL
LIN {X 0,Y 460.501,Z 627.246,A -85,B 0,C 180,E1 -8146.625,E2 -8146.625} C_VEL
LIN {X 0,Y 460.526,Z 627.246,A -85,B 0,C 180,E1 -8149.734,E2 -8149.734} C_VEL
LIN {X 0,Y 460.502,Z 627.247,A -85,B 0,C 180,E1 -8152.524,E2 -8152.524} C_VEL
LIN {X 0,Y 460.539,Z 627.244,A -85,B 0,C 180,E1 -8155.623,E2 -8155.623} C_VEL
LIN {X 0,Y 460.507,Z 627.247,A -85,B 0,C 180,E1 -8158.742,E2 -8158.742} C_VEL
LIN {X 0,Y 460.553,Z 627.303,A -85,B 0,C 180,E1 -8161.02,E2 -8161.02} C_VEL
LIN {X 0,Y 462.692,Z 637.939,A -85,B 0,C 180,E1 -8163.318,E2 -8163.318} C_VEL
LIN {X 0,Y 462.834,Z 641.666,A -85,B 0,C 180,E1 -8164.069,E2 -8164.069} C_VEL
LIN {X 0,Y 466.893,Z 659.81,A -85,B 0,C 180,E1 -8164.578,E2 -8164.578} C_VEL
LIN {X 0,Y 466.209,Z 733.515,A -85,B 0,C 180,E1 -8165.738,E2 -8165.738} C_VEL
LIN {X 0,Y 465.563,Z 739.36,A -85,B 0,C 180,E1 -8165.802,E2 -8165.802} C_VEL
LIN {X 0,Y 459.969,Z 758.393,A -85,B 0,C 180,E1 -8165.853,E2 -8165.853} C_VEL
LIN {X 0,Y 459.267,Z 764.241,A -85,B 0,C 180,E1 -8165.916,E2 -8165.916} C_VEL
LIN {X 0,Y 458.986,Z 781.61,A -85,B 0,C 180,E1 -8166.241,E2 -8166.241} C_VEL
LIN {X 0,Y 458.526,Z 796.2,A -85,B 0,C 180,E1 -8166.698,E2 -8166.698} C_VEL
LIN {X 0,Y 458.02,Z 808.449,A -85,B 0,C 180,E1 -8167.243,E2 -8167.243} C_VEL
LIN {X 0,Y 457.304,Z 821.558,A -85,B 0,C 180,E1 -8168,E2 -8168} C_VEL
LIN {X 0,Y 456.616,Z 833.951,A -85,B 0,C 180,E1 -8168.914,E2 -8168.914} C_VEL
LIN {X 0,Y 455.855,Z 845.252,A -85,B 0,C 180,E1 -8169.938,E2 -8169.938} C_VEL
LIN {X 0,Y 455.141,Z 855.621,A -85,B 0,C 180,E1 -8171.079,E2 -8171.079} C_VEL
LIN {X 0,Y 454.414,Z 865.869,A -85,B 0,C 180,E1 -8172.447,E2 -8172.447} C_VEL
LIN {X 0,Y 453.902,Z 874.328,A -85,B 0,C 180,E1 -8173.817,E2 -8173.817} C_VEL
LIN {X 0,Y 453.317,Z 882.368,A -85,B 0,C 180,E1 -8175.408,E2 -8175.408} C_VEL
LIN {X 0,Y 452.978,Z 888.812,A -85,B 0,C 180,E1 -8176.999,E2 -8176.999} C_VEL
LIN {X 0,Y 452.693,Z 894.496,A -85,B 0,C 180,E1 -8178.81,E2 -8178.81} C_VEL
LIN {X 0,Y 452.545,Z 897.706,A -85,B 0,C 180,E1 -8180.164,E2 -8180.164} C_VEL
LIN {X 0,Y 452.496,Z 900.687,A -85,B 0,C 180,E1 -8181.965,E2 -8181.965} C_VEL
LIN {X 0,Y 452.518,Z 902.293,A -85,B 0,C 180,E1 -8183.759,E2 -8183.759} C_VEL
LIN {X 0,Y 452.427,Z 902.579,A -85,B 0,C 180,E1 -8185.545,E2 -8185.545} C_VEL
LIN {X 0,Y 452.505,Z 901.547,A -85,B 0,C 180,E1 -8187.329,E2 -8187.329} C_VEL
LIN {X 0,Y 452.495,Z 899.2,A -85,B 0,C 180,E1 -8189.11,E2 -8189.11} C_VEL
LIN {X 0,Y 452.54,Z 895.478,A -85,B 0,C 180,E1 -8190.89,E2 -8190.89} C_VEL
LIN {X 0,Y 452.828,Z 890.238,A -85,B 0,C 180,E1 -8192.669,E2 -8192.669} C_VEL
LIN {X 0,Y 453.193,Z 885.195,A -85,B 0,C 180,E1 -8194.002,E2 -8194.002} C_VEL
LIN {X 0,Y 453.691,Z 878.004,A -85,B 0,C 180,E1 -8195.556,E2 -8195.556} C_VEL
LIN {X 0,Y 454.109,Z 870.488,A -85,B 0,C 180,E1 -8196.889,E2 -8196.889} C_VEL
LIN {X 0,Y 454.662,Z 861.159,A -85,B 0,C 180,E1 -8198.266,E2 -8198.266} C_VEL
LIN {X 0,Y 455.464,Z 850.555,A -85,B 0,C 180,E1 -8199.548,E2 -8199.548} C_VEL
LIN {X 0,Y 456.239,Z 839.418,A -85,B 0,C 180,E1 -8200.653,E2 -8200.653} C_VEL
LIN {X 0,Y 456.883,Z 827.143,A -85,B 0,C 180,E1 -8201.648,E2 -8201.648} C_VEL
LIN {X 0,Y 457.581,Z 815.3,A -85,B 0,C 180,E1 -8202.417,E2 -8202.417} C_VEL
LIN {X 0,Y 458.201,Z 802.349,A -85,B 0,C 180,E1 -8203.076,E2 -8203.076} C_VEL
LIN {X 0,Y 458.583,Z 789.323,A -85,B 0,C 180,E1 -8203.572,E2 -8203.572} C_VEL
LIN {X 0,Y 458.864,Z 775.244,A -85,B 0,C 180,E1 -8203.931,E2 -8203.931} C_VEL
LIN {X 0,Y 460.187,Z 661.188,A -85,B 0,C 180,E1 -8205.735,E2 -8205.735} C_VEL
LIN {X 0,Y 455.864,Z 641.846,A -85,B 0,C 180,E1 -8206.258,E2 -8206.258} C_VEL
LIN {X 0,Y 455.307,Z 636.845,A -85,B 0,C 180,E1 -8207.286,E2 -8207.286} C_VEL
LIN {X 0,Y 453.543,Z 628.119,A -85,B 0,C 180,E1 -8209.202,E2 -8209.202} C_VEL
LIN {X 0,Y 453.48,Z 628.126,A -85,B 0,C 180,E1 -8212.796,E2 -8212.796} C_VEL
LIN {X 0,Y 453.469,Z 628.123,A -85,B 0,C 180,E1 -8215.985,E2 -8215.985} C_VEL
LIN {X 0,Y 453.462,Z 628.126,A -85,B 0,C 180,E1 -8218.715,E2 -8218.715} C_VEL
LIN {X 0,Y 453.438,Z 628.125,A -85,B 0,C 180,E1 -8221.802,E2 -8221.802} C_VEL
LIN {X 0,Y 453.472,Z 628.127,A -85,B 0,C 180,E1 -8224.99,E2 -8224.99} C_VEL
LIN {X 0,Y 453.451,Z 628.124,A -85,B 0,C 180,E1 -8228.313,E2 -8228.313} C_VEL
LIN {X 0,Y 453.473,Z 628.114,A -85,B 0,C 180,E1 -8230.611,E2 -8230.611} C_VEL
LIN {X 0,Y 453.484,Z 628.118,A -85,B 0,C 180,E1 -8234.528,E2 -8234.528} C_VEL
LIN {X 0,Y 453.439,Z 628.123,A -85,B 0,C 180,E1 -8238.071,E2 -8238.071} C_VEL
LIN {X 0,Y 453.442,Z 628.126,A -85,B 0,C 180,E1 -8240.802,E2 -8240.802} C_VEL
LIN {X 0,Y 453.451,Z 628.115,A -85,B 0,C 180,E1 -8243.916,E2 -8243.916} C_VEL
LIN {X 0,Y 453.482,Z 628.125,A -85,B 0,C 180,E1 -8247.151,E2 -8247.151} C_VEL
LIN {X 0,Y 453.469,Z 628.114,A -85,B 0,C 180,E1 -8250.267,E2 -8250.267} C_VEL
LIN {X 0,Y 453.456,Z 628.129,A -85,B 0,C 180,E1 -8253.29,E2 -8253.29} C_VEL
LIN {X 0,Y 453.495,Z 628.11,A -85,B 0,C 180,E1 -8256.238,E2 -8256.238} C_VEL
LIN {X 0,Y 453.486,Z 628.121,A -85,B 0,C 180,E1 -8259.117,E2 -8259.117} C_VEL
LIN {X 0,Y 453.506,Z 628.108,A -85,B 0,C 180,E1 -8261.944,E2 -8261.944} C_VEL
LIN {X 0,Y 453.543,Z 628.109,A -85,B 0,C 180,E1 -8264.726,E2 -8264.726} C_VEL
LIN {X 0,Y 453.562,Z 628.103,A -85,B 0,C 180,E1 -8268.379,E2 -8268.379} C_VEL
LIN {X 0,Y 453.588,Z 628.101,A -85,B 0,C 180,E1 -8271.086,E2 -8271.086} C_VEL
LIN {X 0,Y 453.647,Z 628.103,A -85,B 0,C 180,E1 -8273.774,E2 -8273.774} C_VEL
LIN {X 0,Y 453.739,Z 628.087,A -85,B 0,C 180,E1 -8277.336,E2 -8277.336} C_VEL
LIN {X 0,Y 453.825,Z 628.077,A -85,B 0,C 180,E1 -8280,E2 -8280} C_VEL
LIN {X 0,Y 453.746,Z 628.085,A -85,B 0,C 180,E1 -8282.663,E2 -8282.663} C_VEL
LIN {X 0,Y 453.655,Z 628.099,A -85,B 0,C 180,E1 -8286.225,E2 -8286.225} C_VEL
LIN {X 0,Y 453.594,Z 628.104,A -85,B 0,C 180,E1 -8288.913,E2 -8288.913} C_VEL
LIN {X 0,Y 453.566,Z 628.109,A -85,B 0,C 180,E1 -8292.529,E2 -8292.529} C_VEL
LIN {X 0,Y 453.559,Z 628.113,A -85,B 0,C 180,E1 -8296.195,E2 -8296.195} C_VEL
LIN {X 0,Y 453.523,Z 628.11,A -85,B 0,C 180,E1 -8299.041,E2 -8299.041} C_VEL
LIN {X 0,Y 453.479,Z 628.121,A -85,B 0,C 180,E1 -8301.836,E2 -8301.836} C_VEL
LIN {X 0,Y 453.503,Z 628.116,A -85,B 0,C 180,E1 -8304.735,E2 -8304.735} C_VEL
LIN {X 0,Y 453.534,Z 628.113,A -85,B 0,C 180,E1 -8307.959,E2 -8307.959} C_VEL
LIN {X 0,Y 453.468,Z 628.119,A -85,B 0,C 180,E1 -8311.525,E2 -8311.525} C_VEL
LIN {X 0,Y 453.489,Z 628.121,A -85,B 0,C 180,E1 -8314.777,E2 -8314.777} C_VEL
LIN {X 0,Y 453.482,Z 628.125,A -85,B 0,C 180,E1 -8318.31,E2 -8318.31} C_VEL
LIN {X 0,Y 453.517,Z 628.12,A -85,B 0,C 180,E1 -8320.606,E2 -8320.606} C_VEL
LIN {X 0,Y 453.468,Z 628.124,A -85,B 0,C 180,E1 -8324.221,E2 -8324.221} C_VEL
LIN {X 0,Y 453.47,Z 628.121,A -85,B 0,C 180,E1 -8327.006,E2 -8327.006} C_VEL
LIN {X 0,Y 453.519,Z 628.12,A -85,B 0,C 180,E1 -8330.553,E2 -8330.553} C_VEL
LIN {X 0,Y 453.459,Z 628.123,A -85,B 0,C 180,E1 -8333.917,E2 -8333.917} C_VEL
LIN {X 0,Y 453.485,Z 628.123,A -85,B 0,C 180,E1 -8337.151,E2 -8337.151} C_VEL
LIN {X 0,Y 453.525,Z 628.119,A -85,B 0,C 180,E1 -8340.782,E2 -8340.782} C_VEL
LIN {X 0,Y 453.527,Z 628.249,A -85,B 0,C 180,E1 -8341.131,E2 -8341.131} C_VEL
LIN {X 0,Y 456.776,Z 642.652,A -85,B 0,C 180,E1 -8343.746,E2 -8343.746} C_VEL
LIN {X 0,Y 457.349,Z 647.106,A -85,B 0,C 180,E1 -8344.515,E2 -8344.515} C_VEL
LIN {X 0,Y 456.07,Z 669.358,A -85,B 0,C 180,E1 -8348.104,E2 -8348.104} C_VEL
LIN {X 0,Y 455.857,Z 673.716,A -85,B 0,C 180,E1 -8348.773,E2 -8348.773} C_VEL
LIN {X 0,Y 460,Z 697.841,A -85,B 0,C 180,E1 -8349.351,E2 -8349.351} C_VEL
LIN {X 0,Y 458.669,Z 812.214,A -85,B 0,C 180,E1 -8351.172,E2 -8351.172} C_VEL
LIN {X 0,Y 458.184,Z 826.756,A -85,B 0,C 180,E1 -8351.586,E2 -8351.586} C_VEL
LIN {X 0,Y 457.635,Z 840.663,A -85,B 0,C 180,E1 -8352.168,E2 -8352.168} C_VEL
LIN {X 0,Y 456.926,Z 854.203,A -85,B 0,C 180,E1 -8352.926,E2 -8352.926} C_VEL
LIN {X 0,Y 456.225,Z 866.3,A -85,B 0,C 180,E1 -8353.787,E2 -8353.787} C_VEL
LIN {X 0,Y 455.438,Z 877.806,A -85,B 0,C 180,E1 -8354.791,E2 -8354.791} C_VEL
LIN {X 0,Y 454.738,Z 888.377,A -85,B 0,C 180,E1 -8355.912,E2 -8355.912} C_VEL
LIN {X 0,Y 454.086,Z 898.306,A -85,B 0,C 180,E1 -8357.179,E2 -8357.179} C_VEL
LIN {X 0,Y 453.598,Z 907.556,A -85,B 0,C 180,E1 -8358.606,E2 -8358.606} C_VEL
LIN {X 0,Y 453.104,Z 915.858,A -85,B 0,C 180,E1 -8360.176,E2 -8360.176} C_VEL
LIN {X 0,Y 452.838,Z 921.664,A -85,B 0,C 180,E1 -8361.521,E2 -8361.521} C_VEL
LIN {X 0,Y 452.657,Z 926.425,A -85,B 0,C 180,E1 -8362.865,E2 -8362.865} C_VEL
LIN {X 0,Y 452.578,Z 931.359,A -85,B 0,C 180,E1 -8364.654,E2 -8364.654} C_VEL
LIN {X 0,Y 452.475,Z 934.785,A -85,B 0,C 180,E1 -8366.438,E2 -8366.438} C_VEL
LIN {X 0,Y 452.45,Z 936.812,A -85,B 0,C 180,E1 -8368.22,E2 -8368.22} C_VEL
LIN {X 0,Y 452.462,Z 937.483,A -85,B 0,C 180,E1 -8370,E2 -8370} C_VEL
LIN {X 0,Y 452.45,Z 936.808,A -85,B 0,C 180,E1 -8371.78,E2 -8371.78} C_VEL
LIN {X 0,Y 452.475,Z 934.778,A -85,B 0,C 180,E1 -8373.562,E2 -8373.562} C_VEL
LIN {X 0,Y 452.577,Z 931.348,A -85,B 0,C 180,E1 -8375.346,E2 -8375.346} C_VEL
LIN {X 0,Y 452.656,Z 926.412,A -85,B 0,C 180,E1 -8377.135,E2 -8377.135} C_VEL
LIN {X 0,Y 452.927,Z 919.834,A -85,B 0,C 180,E1 -8378.927,E2 -8378.927} C_VEL
LIN {X 0,Y 453.25,Z 912.524,A -85,B 0,C 180,E1 -8380.497,E2 -8380.497} C_VEL
LIN {X 0,Y 453.758,Z 904.876,A -85,B 0,C 180,E1 -8381.842,E2 -8381.842} C_VEL
LIN {X 0,Y 454.326,Z 895.425,A -85,B 0,C 180,E1 -8383.229,E2 -8383.229} C_VEL
LIN {X 0,Y 455.023,Z 884.616,A -85,B 0,C 180,E1 -8384.536,E2 -8384.536} C_VEL
LIN {X 0,Y 455.759,Z 873.313,A -85,B 0,C 180,E1 -8385.656,E2 -8385.656} C_VEL
LIN {X 0,Y 456.607,Z 860.838,A -85,B 0,C 180,E1 -8386.659,E2 -8386.659} C_VEL
LIN {X 0,Y 457.377,Z 847.529,A -85,B 0,C 180,E1 -8387.51,E2 -8387.51} C_VEL
LIN {X 0,Y 458.001,Z 834.35,A -85,B 0,C 180,E1 -8388.161,E2 -8388.161} C_VEL
LIN {X 0,Y 458.567,Z 820.505,A -85,B 0,C 180,E1 -8388.659,E2 -8388.659} C_VEL
LIN {X 0,Y 458.924,Z 806.258,A -85,B 0,C 180,E1 -8388.991,E2 -8388.991} C_VEL
LIN {X 0,Y 460.184,Z 697.869,A -85,B 0,C 180,E1 -8390.711,E2 -8390.711} C_VEL
LIN {X 0,Y 455.934,Z 673.393,A -85,B 0,C 180,E1 -8391.333,E2 -8391.333} C_VEL
LIN {X 0,Y 457.121,Z 653.801,A -85,B 0,C 180,E1 -8394.526,E2 -8394.526} C_VEL
LIN {X 0,Y 457.489,Z 646.593,A -85,B 0,C 180,E1 -8395.72,E2 -8395.72} C_VEL
LIN {X 0,Y 455.472,Z 636.47,A -85,B 0,C 180,E1 -8397.575,E2 -8397.575} C_VEL
LIN {X 0,Y 453.511,Z 628.122,A -85,B 0,C 180,E1 -8399.187,E2 -8399.187} C_VEL
LIN {X 0,Y 453.466,Z 628.122,A -85,B 0,C 180,E1 -8401.799,E2 -8401.799} C_VEL
LIN {X 0,Y 453.483,Z 628.118,A -85,B 0,C 180,E1 -8404.989,E2 -8404.989} C_VEL
LIN {X 0,Y 453.477,Z 628.119,A -85,B 0,C 180,E1 -8408.31,E2 -8408.31} C_VEL
LIN {X 0,Y 453.515,Z 628.111,A -85,B 0,C 180,E1 -8410.607,E2 -8410.607} C_VEL
LIN {X 0,Y 453.474,Z 628.117,A -85,B 0,C 180,E1 -8414.22,E2 -8414.22} C_VEL
LIN {X 0,Y 453.464,Z 628.122,A -85,B 0,C 180,E1 -8417.005,E2 -8417.005} C_VEL
LIN {X 0,Y 453.532,Z 628.112,A -85,B 0,C 180,E1 -8420.555,E2 -8420.555} C_VEL
LIN {X 0,Y 453.458,Z 628.123,A -85,B 0,C 180,E1 -8423.918,E2 -8423.918} C_VEL
LIN {X 0,Y 453.484,Z 628.117,A -85,B 0,C 180,E1 -8427.151,E2 -8427.151} C_VEL
LIN {X 0,Y 453.476,Z 628.119,A -85,B 0,C 180,E1 -8430.269,E2 -8430.269} C_VEL
LIN {X 0,Y 453.51,Z 628.115,A -85,B 0,C 180,E1 -8433.294,E2 -8433.294} C_VEL
LIN {X 0,Y 453.505,Z 628.116,A -85,B 0,C 180,E1 -8436.239,E2 -8436.239} C_VEL
LIN {X 0,Y 453.484,Z 628.117,A -85,B 0,C 180,E1 -8439.118,E2 -8439.118} C_VEL
LIN {X 0,Y 453.514,Z 628.116,A -85,B 0,C 180,E1 -8441.945,E2 -8441.945} C_VEL
LIN {X 0,Y 453.551,Z 628.109,A -85,B 0,C 180,E1 -8444.727,E2 -8444.727} C_VEL
LIN {X 0,Y 453.562,Z 628.113,A -85,B 0,C 180,E1 -8448.379,E2 -8448.379} C_VEL
LIN {X 0,Y 453.654,Z 628.097,A -85,B 0,C 180,E1 -8451.985,E2 -8451.985} C_VEL
LIN {X 0,Y 453.671,Z 628.093,A -85,B 0,C 180,E1 -8454.667,E2 -8454.667} C_VEL
LIN {X 0,Y 453.746,Z 628.084,A -85,B 0,C 180,E1 -8457.337,E2 -8457.337} C_VEL
LIN {X 0,Y 453.825,Z 628.078,A -85,B 0,C 180,E1 -8460,E2 -8460} C_VEL
LIN {X 0,Y 453.746,Z 628.09,A -85,B 0,C 180,E1 -8462.664,E2 -8462.664} C_VEL
LIN {X 0,Y 453.671,Z 628.094,A -85,B 0,C 180,E1 -8466.226,E2 -8466.226} C_VEL
LIN {X 0,Y 453.593,Z 628.105,A -85,B 0,C 180,E1 -8468.914,E2 -8468.914} C_VEL
LIN {X 0,Y 453.566,Z 628.114,A -85,B 0,C 180,E1 -8472.529,E2 -8472.529} C_VEL
LIN {X 0,Y 453.546,Z 628.11,A -85,B 0,C 180,E1 -8476.196,E2 -8476.196} C_VEL
LIN {X 0,Y 453.519,Z 628.113,A -85,B 0,C 180,E1 -8479.04,E2 -8479.04} C_VEL
LIN {X 0,Y 453.479,Z 628.119,A -85,B 0,C 180,E1 -8481.836,E2 -8481.836} C_VEL
LIN {X 0,Y 453.507,Z 628.119,A -85,B 0,C 180,E1 -8484.735,E2 -8484.735} C_VEL
LIN {X 0,Y 453.508,Z 628.108,A -85,B 0,C 180,E1 -8487.954,E2 -8487.954} C_VEL
LIN {X 0,Y 453.477,Z 628.116,A -85,B 0,C 180,E1 -8490.76,E2 -8490.76} C_VEL
LIN {X 0,Y 453.47,Z 628.117,A -85,B 0,C 180,E1 -8493.914,E2 -8493.914} C_VEL
LIN {X 0,Y 453.454,Z 628.127,A -85,B 0,C 180,E1 -8497.19,E2 -8497.19} C_VEL
LIN {X 0,Y 453.472,Z 628.117,A -85,B 0,C 180,E1 -8500.612,E2 -8500.612} C_VEL
LIN {X 0,Y 453.461,Z 628.122,A -85,B 0,C 180,E1 -8504.222,E2 -8504.222} C_VEL
LIN {X 0,Y 453.428,Z 628.131,A -85,B 0,C 180,E1 -8507.001,E2 -8507.001} C_VEL
LIN {X 0,Y 453.473,Z 628.127,A -85,B 0,C 180,E1 -8509.413,E2 -8509.413} C_VEL
LIN {X 0,Y 453.455,Z 628.126,A -85,B 0,C 180,E1 -8512.811,E2 -8512.811} C_VEL
LIN {X 0,Y 453.469,Z 628.12,A -85,B 0,C 180,E1 -8516.087,E2 -8516.087} C_VEL
LIN {X 0,Y 453.46,Z 628.127,A -85,B 0,C 180,E1 -8519.239,E2 -8519.239} C_VEL
LIN {X 0,Y 453.493,Z 628.127,A -85,B 0,C 180,E1 -8520.716,E2 -8520.716} C_VEL
LIN {X 0,Y 455.78,Z 639.393,A -85,B 0,C 180,E1 -8523.191,E2 -8523.191} C_VEL
LIN {X 0,Y 456,Z 641.962,A -85,B 0,C 180,E1 -8523.724,E2 -8523.724} C_VEL
LIN {X 0,Y 460.305,Z 660.846,A -85,B 0,C 180,E1 -8524.267,E2 -8524.267} C_VEL
LIN {X 0,Y 459.267,Z 764.241,A -85,B 0,C 180,E1 -8525.916,E2 -8525.916} C_VEL
LIN {X 0,Y 458.523,Z 770.097,A -85,B 0,C 180,E1 -8525.977,E2 -8525.977} C_VEL
LIN {X 0,Y 455.565,Z 779.592,A -85,B 0,C 180,E1 -8526.029,E2 -8526.029} C_VEL
LIN {X 0,Y 452.633,Z 788.985,A -85,B 0,C 180,E1 -8526.159,E2 -8526.159} C_VEL
LIN {X 0,Y 452.022,Z 792.789,A -85,B 0,C 180,E1 -8526.263,E2 -8526.263} C_VEL
LIN {X 0,Y 451.95,Z 794.666,A -85,B 0,C 180,E1 -8526.333,E2 -8526.333} C_VEL
LIN {X 0,Y 451.34,Z 808.378,A -85,B 0,C 180,E1 -8526.935,E2 -8526.935} C_VEL
LIN {X 0,Y 450.619,Z 820.85,A -85,B 0,C 180,E1 -8527.656,E2 -8527.656} C_VEL
LIN {X 0,Y 449.855,Z 833.422,A -85,B 0,C 180,E1 -8528.581,E2 -8528.581} C_VEL
LIN {X 0,Y 449.085,Z 844.863,A -85,B 0,C 180,E1 -8529.623,E2 -8529.623} C_VEL
LIN {X 0,Y 448.309,Z 855.342,A -85,B 0,C 180,E1 -8530.779,E2 -8530.779} C_VEL
LIN {X 0,Y 447.548,Z 865.715,A -85,B 0,C 180,E1 -8532.169,E2 -8532.169} C_VEL
LIN {X 0,Y 446.987,Z 874.244,A -85,B 0,C 180,E1 -8533.56,E2 -8533.56} C_VEL
LIN {X 0,Y 446.355,Z 882.348,A -85,B 0,C 180,E1 -8535.175,E2 -8535.175} C_VEL
LIN {X 0,Y 445.959,Z 888.847,A -85,B 0,C 180,E1 -8536.791,E2 -8536.791} C_VEL
LIN {X 0,Y 445.632,Z 894.584,A -85,B 0,C 180,E1 -8538.631,E2 -8538.631} C_VEL
LIN {X 0,Y 445.48,Z 897.846,A -85,B 0,C 180,E1 -8540.006,E2 -8540.006} C_VEL
LIN {X 0,Y 445.426,Z 900.875,A -85,B 0,C 180,E1 -8541.836,E2 -8541.836} C_VEL
LIN {X 0,Y 445.435,Z 902.565,A -85,B 0,C 180,E1 -8543.727,E2 -8543.727} C_VEL
LIN {X 0,Y 445.349,Z 902.864,A -85,B 0,C 180,E1 -8545.474,E2 -8545.474} C_VEL
LIN {X 0,Y 445.43,Z 901.88,A -85,B 0,C 180,E1 -8547.287,E2 -8547.287} C_VEL
LIN {X 0,Y 445.431,Z 899.58,A -85,B 0,C 180,E1 -8549.096,E2 -8549.096} C_VEL
LIN {X 0,Y 445.476,Z 895.908,A -85,B 0,C 180,E1 -8550.904,E2 -8550.904} C_VEL
LIN {X 0,Y 445.779,Z 890.74,A -85,B 0,C 180,E1 -8552.711,E2 -8552.711} C_VEL
LIN {X 0,Y 446.158,Z 885.731,A -85,B 0,C 180,E1 -8554.065,E2 -8554.065} C_VEL
LIN {X 0,Y 446.671,Z 878.598,A -85,B 0,C 180,E1 -8555.644,E2 -8555.644} C_VEL
LIN {X 0,Y 447.103,Z 871.147,A -85,B 0,C 180,E1 -8556.997,E2 -8556.997} C_VEL
LIN {X 0,Y 447.685,Z 862.033,A -85,B 0,C 180,E1 -8558.375,E2 -8558.375} C_VEL
LIN {X 0,Y 448.536,Z 851.391,A -85,B 0,C 180,E1 -8559.697,E2 -8559.697} C_VEL
LIN {X 0,Y 449.318,Z 840.393,A -85,B 0,C 180,E1 -8560.819,E2 -8560.819} C_VEL
LIN {X 0,Y 450.004,Z 828.285,A -85,B 0,C 180,E1 -8561.829,E2 -8561.829} C_VEL
LIN {X 0,Y 450.815,Z 814.702,A -85,B 0,C 180,E1 -8562.721,E2 -8562.721} C_VEL
LIN {X 0,Y 451.454,Z 801.476,A -85,B 0,C 180,E1 -8563.389,E2 -8563.389} C_VEL
LIN {X 0,Y 451.868,Z 787.967,A -85,B 0,C 180,E1 -8563.893,E2 -8563.893} C_VEL
LIN {X 0,Y 452.14,Z 774.313,A -85,B 0,C 180,E1 -8564.228,E2 -8564.228} C_VEL
LIN {X 0,Y 453.513,Z 662.724,A -85,B 0,C 180,E1 -8566.014,E2 -8566.014} C_VEL
LIN {X 0,Y 448.939,Z 642.059,A -85,B 0,C 180,E1 -8566.591,E2 -8566.591} C_VEL
LIN {X 0,Y 447.084,Z 631.896,A -85,B 0,C 180,E1 -8568.767,E2 -8568.767} C_VEL
LIN {X 0,Y 446.493,Z 628.997,A -85,B 0,C 180,E1 -8569.422,E2 -8569.422} C_VEL
LIN {X 0,Y 446.421,Z 629.004,A -85,B 0,C 180,E1 -8572.2,E2 -8572.2} C_VEL
LIN {X 0,Y 446.416,Z 629.004,A -85,B 0,C 180,E1 -8575.155,E2 -8575.155} C_VEL
LIN {X 0,Y 446.419,Z 629.003,A -85,B 0,C 180,E1 -8578.183,E2 -8578.183} C_VEL
LIN {X 0,Y 446.393,Z 629.005,A -85,B 0,C 180,E1 -8581.302,E2 -8581.302} C_VEL
LIN {X 0,Y 446.417,Z 629.003,A -85,B 0,C 180,E1 -8584.524,E2 -8584.524} C_VEL
LIN {X 0,Y 446.403,Z 629.001,A -85,B 0,C 180,E1 -8588.076,E2 -8588.076} C_VEL
LIN {X 0,Y 446.403,Z 629.003,A -85,B 0,C 180,E1 -8591.394,E2 -8591.394} C_VEL
LIN {X 0,Y 446.452,Z 629.001,A -85,B 0,C 180,E1 -8595.104,E2 -8595.104} C_VEL
LIN {X 0,Y 446.403,Z 629.002,A -85,B 0,C 180,E1 -8598.605,E2 -8598.605} C_VEL
LIN {X 0,Y 446.406,Z 628.988,A -85,B 0,C 180,E1 -8601.923,E2 -8601.923} C_VEL
LIN {X 0,Y 446.425,Z 629.002,A -85,B 0,C 180,E1 -8605.476,E2 -8605.476} C_VEL
LIN {X 0,Y 446.418,Z 628.998,A -85,B 0,C 180,E1 -8608.699,E2 -8608.699} C_VEL
LIN {X 0,Y 446.45,Z 628.996,A -85,B 0,C 180,E1 -8611.83,E2 -8611.83} C_VEL
LIN {X 0,Y 446.432,Z 628.996,A -85,B 0,C 180,E1 -8614.846,E2 -8614.846} C_VEL
LIN {X 0,Y 446.452,Z 628.993,A -85,B 0,C 180,E1 -8618.245,E2 -8618.245} C_VEL
LIN {X 0,Y 446.455,Z 628.989,A -85,B 0,C 180,E1 -8621.649,E2 -8621.649} C_VEL
LIN {X 0,Y 446.511,Z 628.984,A -85,B 0,C 180,E1 -8624.48,E2 -8624.48} C_VEL
LIN {X 0,Y 446.52,Z 628.981,A -85,B 0,C 180,E1 -8628.193,E2 -8628.193} C_VEL
LIN {X 0,Y 446.536,Z 628.978,A -85,B 0,C 180,E1 -8630.944,E2 -8630.944} C_VEL
LIN {X 0,Y 446.616,Z 628.981,A -85,B 0,C 180,E1 -8633.676,E2 -8633.676} C_VEL
LIN {X 0,Y 446.686,Z 628.965,A -85,B 0,C 180,E1 -8637.294,E2 -8637.294} C_VEL
LIN {X 0,Y 446.794,Z 628.952,A -85,B 0,C 180,E1 -8640,E2 -8640} C_VEL
LIN {X 0,Y 446.693,Z 628.964,A -85,B 0,C 180,E1 -8642.705,E2 -8642.705} C_VEL
LIN {X 0,Y 446.623,Z 628.974,A -85,B 0,C 180,E1 -8646.324,E2 -8646.324} C_VEL
LIN {X 0,Y 446.539,Z 628.983,A -85,B 0,C 180,E1 -8649.055,E2 -8649.055} C_VEL
LIN {X 0,Y 446.524,Z 628.985,A -85,B 0,C 180,E1 -8652.729,E2 -8652.729} C_VEL
LIN {X 0,Y 446.522,Z 628.99,A -85,B 0,C 180,E1 -8656.238,E2 -8656.238} C_VEL
LIN {X 0,Y 446.472,Z 628.988,A -85,B 0,C 180,E1 -8659.303,E2 -8659.303} C_VEL
LIN {X 0,Y 446.421,Z 629.003,A -85,B 0,C 180,E1 -8662.199,E2 -8662.199} C_VEL
LIN {X 0,Y 446.446,Z 628.994,A -85,B 0,C 180,E1 -8665.153,E2 -8665.153} C_VEL
LIN {X 0,Y 446.486,Z 628.993,A -85,B 0,C 180,E1 -8668.178,E2 -8668.178} C_VEL
LIN {X 0,Y 446.421,Z 628.998,A -85,B 0,C 180,E1 -8671.775,E2 -8671.775} C_VEL
LIN {X 0,Y 446.431,Z 629.003,A -85,B 0,C 180,E1 -8674.523,E2 -8674.523} C_VEL
LIN {X 0,Y 446.437,Z 628.999,A -85,B 0,C 180,E1 -8678.082,E2 -8678.082} C_VEL
LIN {X 0,Y 446.445,Z 628.997,A -85,B 0,C 180,E1 -8680.92,E2 -8680.92} C_VEL
LIN {X 0,Y 446.403,Z 629,A -85,B 0,C 180,E1 -8683.846,E2 -8683.846} C_VEL
LIN {X 0,Y 446.422,Z 629,A -85,B 0,C 180,E1 -8686.4,E2 -8686.4} C_VEL
LIN {X 0,Y 446.453,Z 628.995,A -85,B 0,C 180,E1 -8689.803,E2 -8689.803} C_VEL
LIN {X 0,Y 446.43,Z 629,A -85,B 0,C 180,E1 -8692.123,E2 -8692.123} C_VEL
LIN {X 0,Y 446.432,Z 628.999,A -85,B 0,C 180,E1 -8695.477,E2 -8695.477} C_VEL
LIN {X 0,Y 446.418,Z 628.997,A -85,B 0,C 180,E1 -8698.7,E2 -8698.7} C_VEL
LIN {X 0,Y 446.512,Z 629.077,A -85,B 0,C 180,E1 -8700.852,E2 -8700.852} C_VEL
LIN {X 0,Y 450.062,Z 645.208,A -85,B 0,C 180,E1 -8703.823,E2 -8703.823} C_VEL
LIN {X 0,Y 450.389,Z 649.448,A -85,B 0,C 180,E1 -8704.555,E2 -8704.555} C_VEL
LIN {X 0,Y 449.123,Z 670.127,A -85,B 0,C 180,E1 -8707.941,E2 -8707.941} C_VEL
LIN {X 0,Y 448.91,Z 673.216,A -85,B 0,C 180,E1 -8708.442,E2 -8708.442} C_VEL
LIN {X 0,Y 453.284,Z 698.021,A -85,B 0,C 180,E1 -8709.057,E2 -8709.057} C_VEL
LIN {X 0,Y 451.944,Z 811.284,A -85,B 0,C 180,E1 -8710.881,E2 -8710.881} C_VEL
LIN {X 0,Y 451.446,Z 826.063,A -85,B 0,C 180,E1 -8711.301,E2 -8711.301} C_VEL
LIN {X 0,Y 450.892,Z 838.989,A -85,B 0,C 180,E1 -8711.836,E2 -8711.836} C_VEL
LIN {X 0,Y 450.168,Z 852.677,A -85,B 0,C 180,E1 -8712.594,E2 -8712.594} C_VEL
LIN {X 0,Y 449.334,Z 865.846,A -85,B 0,C 180,E1 -8713.531,E2 -8713.531} C_VEL
LIN {X 0,Y 448.538,Z 877.391,A -85,B 0,C 180,E1 -8714.552,E2 -8714.552} C_VEL
LIN {X 0,Y 447.782,Z 887.989,A -85,B 0,C 180,E1 -8715.688,E2 -8715.688} C_VEL
LIN {X 0,Y 447.05,Z 898.719,A -85,B 0,C 180,E1 -8717.082,E2 -8717.082} C_VEL
LIN {X 0,Y 446.587,Z 907.216,A -85,B 0,C 180,E1 -8718.425,E2 -8718.425} C_VEL
LIN {X 0,Y 446.032,Z 915.537,A -85,B 0,C 180,E1 -8720.019,E2 -8720.019} C_VEL
LIN {X 0,Y 445.783,Z 921.355,A -85,B 0,C 180,E1 -8721.386,E2 -8721.386} C_VEL
LIN {X 0,Y 445.582,Z 926.126,A -85,B 0,C 180,E1 -8722.751,E2 -8722.751} C_VEL
LIN {X 0,Y 445.49,Z 931.069,A -85,B 0,C 180,E1 -8724.568,E2 -8724.568} C_VEL
LIN {X 0,Y 445.375,Z 934.502,A -85,B 0,C 180,E1 -8726.381,E2 -8726.381} C_VEL
LIN {X 0,Y 445.368,Z 936.535,A -85,B 0,C 180,E1 -8728.191,E2 -8728.191} C_VEL
LIN {X 0,Y 445.368,Z 937.21,A -85,B 0,C 180,E1 -8730,E2 -8730} C_VEL
LIN {X 0,Y 445.367,Z 936.54,A -85,B 0,C 180,E1 -8731.808,E2 -8731.808} C_VEL
LIN {X 0,Y 445.374,Z 934.514,A -85,B 0,C 180,E1 -8733.619,E2 -8733.619} C_VEL
LIN {X 0,Y 445.489,Z 931.09,A -85,B 0,C 180,E1 -8735.431,E2 -8735.431} C_VEL
LIN {X 0,Y 445.582,Z 926.162,A -85,B 0,C 180,E1 -8737.249,E2 -8737.249} C_VEL
LIN {X 0,Y 445.865,Z 919.597,A -85,B 0,C 180,E1 -8739.069,E2 -8739.069} C_VEL
LIN {X 0,Y 446.228,Z 912.301,A -85,B 0,C 180,E1 -8740.665,E2 -8740.665} C_VEL
LIN {X 0,Y 446.824,Z 903.29,A -85,B 0,C 180,E1 -8742.259,E2 -8742.259} C_VEL
LIN {X 0,Y 447.443,Z 893.844,A -85,B 0,C 180,E1 -8743.627,E2 -8743.627} C_VEL
LIN {X 0,Y 448.181,Z 883.404,A -85,B 0,C 180,E1 -8744.879,E2 -8744.879} C_VEL
LIN {X 0,Y 448.989,Z 871.912,A -85,B 0,C 180,E1 -8746.015,E2 -8746.015} C_VEL
LIN {X 0,Y 449.868,Z 859.193,A -85,B 0,C 180,E1 -8747.033,E2 -8747.033} C_VEL
LIN {X 0,Y 450.696,Z 846.145,A -85,B 0,C 180,E1 -8747.86,E2 -8747.86} C_VEL
LIN {X 0,Y 451.341,Z 833.145,A -85,B 0,C 180,E1 -8748.498,E2 -8748.498} C_VEL
LIN {X 0,Y 451.934,Z 818.939,A -85,B 0,C 180,E1 -8749.002,E2 -8749.002} C_VEL
LIN {X 0,Y 452.287,Z 805.377,A -85,B 0,C 180,E1 -8749.31,E2 -8749.31} C_VEL
LIN {X 0,Y 453.586,Z 698.725,A -85,B 0,C 180,E1 -8751.027,E2 -8751.027} C_VEL
LIN {X 0,Y 449.415,Z 674.976,A -85,B 0,C 180,E1 -8751.644,E2 -8751.644} C_VEL
LIN {X 0,Y 449.098,Z 673.107,A -85,B 0,C 180,E1 -8751.696,E2 -8751.696} C_VEL
LIN {X 0,Y 450.363,Z 653.679,A -85,B 0,C 180,E1 -8754.919,E2 -8754.919} C_VEL
LIN {X 0,Y 450.616,Z 647.92,A -85,B 0,C 180,E1 -8755.893,E2 -8755.893} C_VEL
LIN {X 0,Y 448.201,Z 636.372,A -85,B 0,C 180,E1 -8758.061,E2 -8758.061} C_VEL
LIN {X 0,Y 446.458,Z 628.999,A -85,B 0,C 180,E1 -8759.523,E2 -8759.523} C_VEL
LIN {X 0,Y 446.423,Z 628.997,A -85,B 0,C 180,E1 -8762.361,E2 -8762.361} C_VEL
LIN {X 0,Y 446.423,Z 628.998,A -85,B 0,C 180,E1 -8765.626,E2 -8765.626} C_VEL
LIN {X 0,Y 446.466,Z 628.996,A -85,B 0,C 180,E1 -8769.025,E2 -8769.025} C_VEL
LIN {X 0,Y 446.437,Z 628.997,A -85,B 0,C 180,E1 -8772.278,E2 -8772.278} C_VEL
LIN {X 0,Y 446.455,Z 628.994,A -85,B 0,C 180,E1 -8775.103,E2 -8775.103} C_VEL
LIN {X 0,Y 446.436,Z 628.992,A -85,B 0,C 180,E1 -8778.61,E2 -8778.61} C_VEL
LIN {X 0,Y 446.474,Z 628.993,A -85,B 0,C 180,E1 -8780.976,E2 -8780.976} C_VEL
LIN {X 0,Y 446.423,Z 628.998,A -85,B 0,C 180,E1 -8784.374,E2 -8784.374} C_VEL
LIN {X 0,Y 446.423,Z 628.991,A -85,B 0,C 180,E1 -8787.639,E2 -8787.639} C_VEL
LIN {X 0,Y 446.45,Z 628.992,A -85,B 0,C 180,E1 -8790.791,E2 -8790.791} C_VEL
LIN {X 0,Y 446.478,Z 628.992,A -85,B 0,C 180,E1 -8793.849,E2 -8793.849} C_VEL
LIN {X 0,Y 446.431,Z 628.994,A -85,B 0,C 180,E1 -8796.824,E2 -8796.824} C_VEL
LIN {X 0,Y 446.446,Z 628.999,A -85,B 0,C 180,E1 -8799.737,E2 -8799.737} C_VEL
LIN {X 0,Y 446.467,Z 628.993,A -85,B 0,C 180,E1 -8802.597,E2 -8802.597} C_VEL
LIN {X 0,Y 446.475,Z 628.991,A -85,B 0,C 180,E1 -8805.413,E2 -8805.413} C_VEL
LIN {X 0,Y 446.519,Z 628.993,A -85,B 0,C 180,E1 -8808.193,E2 -8808.193} C_VEL
LIN {X 0,Y 446.602,Z 628.974,A -85,B 0,C 180,E1 -8811.858,E2 -8811.858} C_VEL
LIN {X 0,Y 446.645,Z 628.969,A -85,B 0,C 180,E1 -8814.583,E2 -8814.583} C_VEL
LIN {X 0,Y 446.665,Z 628.974,A -85,B 0,C 180,E1 -8818.197,E2 -8818.197} C_VEL
LIN {X 0,Y 446.794,Z 628.954,A -85,B 0,C 180,E1 -8820,E2 -8820} C_VEL
LIN {X 0,Y 446.693,Z 628.968,A -85,B 0,C 180,E1 -8822.706,E2 -8822.706} C_VEL
LIN {X 0,Y 446.641,Z 628.97,A -85,B 0,C 180,E1 -8826.324,E2 -8826.324} C_VEL
LIN {X 0,Y 446.538,Z 628.983,A -85,B 0,C 180,E1 -8829.056,E2 -8829.056} C_VEL
LIN {X 0,Y 446.524,Z 628.991,A -85,B 0,C 180,E1 -8832.73,E2 -8832.73} C_VEL
LIN {X 0,Y 446.498,Z 628.988,A -85,B 0,C 180,E1 -8836.228,E2 -8836.228} C_VEL
LIN {X 0,Y 446.47,Z 628.989,A -85,B 0,C 180,E1 -8839.304,E2 -8839.304} C_VEL
LIN {X 0,Y 446.421,Z 629,A -85,B 0,C 180,E1 -8842.2,E2 -8842.2} C_VEL
LIN {X 0,Y 446.448,Z 628.998,A -85,B 0,C 180,E1 -8845.153,E2 -8845.153} C_VEL
LIN {X 0,Y 446.451,Z 628.988,A -85,B 0,C 180,E1 -8848.181,E2 -8848.181} C_VEL
LIN {X 0,Y 446.418,Z 629.002,A -85,B 0,C 180,E1 -8851.301,E2 -8851.301} C_VEL
LIN {X 0,Y 446.425,Z 628.997,A -85,B 0,C 180,E1 -8854.524,E2 -8854.524} C_VEL
LIN {X 0,Y 446.414,Z 628.999,A -85,B 0,C 180,E1 -8858.079,E2 -8858.079} C_VEL
LIN {X 0,Y 446.408,Z 628.998,A -85,B 0,C 180,E1 -8861.394,E2 -8861.394} C_VEL
LIN {X 0,Y 446.452,Z 628.995,A -85,B 0,C 180,E1 -8865.104,E2 -8865.104} C_VEL
LIN {X 0,Y 446.404,Z 629.004,A -85,B 0,C 180,E1 -8868.606,E2 -8868.606} C_VEL
LIN {X 0,Y 446.414,Z 629.003,A -85,B 0,C 180,E1 -8871.922,E2 -8871.922} C_VEL
LIN {X 0,Y 446.425,Z 629.004,A -85,B 0,C 180,E1 -8875.477,E2 -8875.477} C_VEL
LIN {X 0,Y 446.412,Z 629.004,A -85,B 0,C 180,E1 -8878.699,E2 -8878.699} C_VEL
LIN {X 0,Y 446.456,Z 629.019,A -85,B 0,C 180,E1 -8880.415,E2 -8880.415} C_VEL
LIN {X 0,Y 448.849,Z 640.552,A -85,B 0,C 180,E1 -8882.994,E2 -8882.994} C_VEL
LIN {X 0,Y 449.126,Z 642.339,A -85,B 0,C 180,E1 -8883.366,E2 -8883.366} C_VEL
LIN {X 0,Y 453.467,Z 660.462,A -85,B 0,C 180,E1 -8883.907,E2 -8883.907} C_VEL
LIN {X 0,Y 453.854,Z 663.247,A -85,B 0,C 180,E1 -8883.974,E2 -8883.974} C_VEL
LIN {X 0,Y 452.507,Z 778.198,A -85,B 0,C 180,E1 -8885.848,E2 -8885.848} C_VEL
LIN {X 0,Y 452.044,Z 792.45,A -85,B 0,C 180,E1 -8886.251,E2 -8886.251} C_VEL
LIN {X 0,Y 451.95,Z 794.666,A -85,B 0,C 180,E1 -8886.333,E2 -8886.333} C_VEL
LIN {X 0,Y 451.183,Z 800.398,A -85,B 0,C 180,E1 -8886.534,E2 -8886.534} C_VEL
LIN {X 0,Y 448.016,Z 809.523,A -85,B 0,C 180,E1 -8886.84,E2 -8886.84} C_VEL
LIN {X 0,Y 444.731,Z 818.386,A -85,B 0,C 180,E1 -8887.217,E2 -8887.217} C_VEL
LIN {X 0,Y 443.762,Z 823.561,A -85,B 0,C 180,E1 -8887.527,E2 -8887.527} C_VEL
LIN {X 0,Y 442.973,Z 835.747,A -85,B 0,C 180,E1 -8888.476,E2 -8888.476} C_VEL
LIN {X 0,Y 442.123,Z 846.803,A -85,B 0,C 180,E1 -8889.53,E2 -8889.53} C_VEL
LIN {X 0,Y 441.338,Z 856.994,A -85,B 0,C 180,E1 -8890.705,E2 -8890.705} C_VEL
LIN {X 0,Y 440.529,Z 867.077,A -85,B 0,C 180,E1 -8892.115,E2 -8892.115} C_VEL
LIN {X 0,Y 439.905,Z 875.705,A -85,B 0,C 180,E1 -8893.582,E2 -8893.582} C_VEL
LIN {X 0,Y 439.279,Z 883.351,A -85,B 0,C 180,E1 -8895.168,E2 -8895.168} C_VEL
LIN {X 0,Y 438.946,Z 888.894,A -85,B 0,C 180,E1 -8896.576,E2 -8896.576} C_VEL
LIN {X 0,Y 438.585,Z 894.682,A -85,B 0,C 180,E1 -8898.445,E2 -8898.445} C_VEL
LIN {X 0,Y 438.428,Z 897.992,A -85,B 0,C 180,E1 -8899.844,E2 -8899.844} C_VEL
LIN {X 0,Y 438.336,Z 901.069,A -85,B 0,C 180,E1 -8901.703,E2 -8901.703} C_VEL
LIN {X 0,Y 438.357,Z 902.768,A -85,B 0,C 180,E1 -8903.556,E2 -8903.556} C_VEL
LIN {X 0,Y 438.274,Z 903.148,A -85,B 0,C 180,E1 -8905.401,E2 -8905.401} C_VEL
LIN {X 0,Y 438.357,Z 902.209,A -85,B 0,C 180,E1 -8907.243,E2 -8907.243} C_VEL
LIN {X 0,Y 438.34,Z 899.956,A -85,B 0,C 180,E1 -8909.081,E2 -8909.081} C_VEL
LIN {X 0,Y 438.413,Z 896.33,A -85,B 0,C 180,E1 -8910.919,E2 -8910.919} C_VEL
LIN {X 0,Y 438.732,Z 891.217,A -85,B 0,C 180,E1 -8912.755,E2 -8912.755} C_VEL
LIN {X 0,Y 439.124,Z 886.254,A -85,B 0,C 180,E1 -8914.13,E2 -8914.13} C_VEL
LIN {X 0,Y 439.653,Z 879.177,A -85,B 0,C 180,E1 -8915.734,E2 -8915.734} C_VEL
LIN {X 0,Y 440.098,Z 871.791,A -85,B 0,C 180,E1 -8917.109,E2 -8917.109} C_VEL
LIN {X 0,Y 440.697,Z 862.832,A -85,B 0,C 180,E1 -8918.497,E2 -8918.497} C_VEL
LIN {X 0,Y 441.584,Z 852.188,A -85,B 0,C 180,E1 -8919.851,E2 -8919.851} C_VEL
LIN {X 0,Y 442.404,Z 841.302,A -85,B 0,C 180,E1 -8920.99,E2 -8920.99} C_VEL
LIN {X 0,Y 443.138,Z 829.375,A -85,B 0,C 180,E1 -8922.015,E2 -8922.015} C_VEL
LIN {X 0,Y 443.985,Z 816.02,A -85,B 0,C 180,E1 -8922.92,E2 -8922.92} C_VEL
LIN {X 0,Y 444.667,Z 803.106,A -85,B 0,C 180,E1 -8923.598,E2 -8923.598} C_VEL
LIN {X 0,Y 445.055,Z 790.161,A -85,B 0,C 180,E1 -8924.11,E2 -8924.11} C_VEL
LIN {X 0,Y 445.407,Z 776.233,A -85,B 0,C 180,E1 -8924.477,E2 -8924.477} C_VEL
LIN {X 0,Y 446.846,Z 663.413,A -85,B 0,C 180,E1 -8926.314,E2 -8926.314} C_VEL
LIN {X 0,Y 442.262,Z 643.771,A -85,B 0,C 180,E1 -8926.866,E2 -8926.866} C_VEL
LIN {X 0,Y 441.886,Z 642.304,A -85,B 0,C 180,E1 -8926.933,E2 -8926.933} C_VEL
LIN {X 0,Y 439.66,Z 630.958,A -85,B 0,C 180,E1 -8929.416,E2 -8929.416} C_VEL
LIN {X 0,Y 439.44,Z 629.875,A -85,B 0,C 180,E1 -8929.685,E2 -8929.685} C_VEL
LIN {X 0,Y 439.366,Z 629.884,A -85,B 0,C 180,E1 -8932.576,E2 -8932.576} C_VEL
LIN {X 0,Y 439.357,Z 629.881,A -85,B 0,C 180,E1 -8935.588,E2 -8935.588} C_VEL
LIN {X 0,Y 439.383,Z 629.879,A -85,B 0,C 180,E1 -8938.676,E2 -8938.676} C_VEL
LIN {X 0,Y 439.346,Z 629.881,A -85,B 0,C 180,E1 -8942.024,E2 -8942.024} C_VEL
LIN {X 0,Y 439.388,Z 629.877,A -85,B 0,C 180,E1 -8945.338,E2 -8945.338} C_VEL
LIN {X 0,Y 439.359,Z 629.882,A -85,B 0,C 180,E1 -8948.598,E2 -8948.598} C_VEL
LIN {X 0,Y 439.351,Z 629.879,A -85,B 0,C 180,E1 -8952.21,E2 -8952.21} C_VEL
LIN {X 0,Y 439.4,Z 629.878,A -85,B 0,C 180,E1 -8955.27,E2 -8955.27} C_VEL
LIN {X 0,Y 439.356,Z 629.884,A -85,B 0,C 180,E1 -8959.016,E2 -8959.016} C_VEL
LIN {X 0,Y 439.343,Z 629.868,A -85,B 0,C 180,E1 -8962.564,E2 -8962.564} C_VEL
LIN {X 0,Y 439.397,Z 629.868,A -85,B 0,C 180,E1 -8964.843,E2 -8964.843} C_VEL
LIN {X 0,Y 439.374,Z 629.874,A -85,B 0,C 180,E1 -8968.139,E2 -8968.139} C_VEL
LIN {X 0,Y 439.405,Z 629.876,A -85,B 0,C 180,E1 -8971.605,E2 -8971.605} C_VEL
LIN {X 0,Y 439.373,Z 629.873,A -85,B 0,C 180,E1 -8974.413,E2 -8974.413} C_VEL
LIN {X 0,Y 439.366,Z 629.878,A -85,B 0,C 180,E1 -8977.424,E2 -8977.424} C_VEL
LIN {X 0,Y 439.444,Z 629.865,A -85,B 0,C 180,E1 -8980.663,E2 -8980.663} C_VEL
LIN {X 0,Y 439.466,Z 629.863,A -85,B 0,C 180,E1 -8984.224,E2 -8984.224} C_VEL
LIN {X 0,Y 439.486,Z 629.859,A -85,B 0,C 180,E1 -8988.001,E2 -8988.001} C_VEL
LIN {X 0,Y 439.507,Z 629.863,A -85,B 0,C 180,E1 -8991.725,E2 -8991.725} C_VEL
LIN {X 0,Y 439.608,Z 629.845,A -85,B 0,C 180,E1 -8994.495,E2 -8994.495} C_VEL
LIN {X 0,Y 439.636,Z 629.846,A -85,B 0,C 180,E1 -8998.168,E2 -8998.168} C_VEL
LIN {X 0,Y 439.764,Z 629.828,A -85,B 0,C 180,E1 -9000,E2 -9000} C_VEL
LIN {X 0,Y 439.642,Z 629.842,A -85,B 0,C 180,E1 -9002.749,E2 -9002.749} C_VEL
LIN {X 0,Y 439.595,Z 629.848,A -85,B 0,C 180,E1 -9006.425,E2 -9006.425} C_VEL
LIN {X 0,Y 439.501,Z 629.86,A -85,B 0,C 180,E1 -9009.201,E2 -9009.201} C_VEL
LIN {X 0,Y 439.468,Z 629.863,A -85,B 0,C 180,E1 -9012.937,E2 -9012.937} C_VEL
LIN {X 0,Y 439.463,Z 629.867,A -85,B 0,C 180,E1 -9016.354,E2 -9016.354} C_VEL
LIN {X 0,Y 439.405,Z 629.87,A -85,B 0,C 180,E1 -9019.626,E2 -9019.626} C_VEL
LIN {X 0,Y 439.366,Z 629.876,A -85,B 0,C 180,E1 -9022.575,E2 -9022.575} C_VEL
LIN {X 0,Y 439.399,Z 629.872,A -85,B 0,C 180,E1 -9025.585,E2 -9025.585} C_VEL
LIN {X 0,Y 439.419,Z 629.873,A -85,B 0,C 180,E1 -9028.673,E2 -9028.673} C_VEL
LIN {X 0,Y 439.372,Z 629.879,A -85,B 0,C 180,E1 -9032.03,E2 -9032.03} C_VEL
LIN {X 0,Y 439.396,Z 629.873,A -85,B 0,C 180,E1 -9035.34,E2 -9035.34} C_VEL
LIN {X 0,Y 439.397,Z 629.877,A -85,B 0,C 180,E1 -9038.593,E2 -9038.593} C_VEL
LIN {X 0,Y 439.4,Z 629.872,A -85,B 0,C 180,E1 -9041.258,E2 -9041.258} C_VEL
LIN {X 0,Y 439.404,Z 629.877,A -85,B 0,C 180,E1 -9044.729,E2 -9044.729} C_VEL
LIN {X 0,Y 439.399,Z 629.872,A -85,B 0,C 180,E1 -9047.796,E2 -9047.796} C_VEL
LIN {X 0,Y 439.438,Z 629.872,A -85,B 0,C 180,E1 -9050.228,E2 -9050.228} C_VEL
LIN {X 0,Y 439.379,Z 629.877,A -85,B 0,C 180,E1 -9053.713,E2 -9053.713} C_VEL
LIN {X 0,Y 439.374,Z 629.882,A -85,B 0,C 180,E1 -9057.054,E2 -9057.054} C_VEL
LIN {X 0,Y 439.447,Z 629.98,A -85,B 0,C 180,E1 -9060.575,E2 -9060.575} C_VEL
LIN {X 0,Y 442.826,Z 645.121,A -85,B 0,C 180,E1 -9063.422,E2 -9063.422} C_VEL
LIN {X 0,Y 443.531,Z 649.532,A -85,B 0,C 180,E1 -9064.217,E2 -9064.217} C_VEL
LIN {X 0,Y 442.271,Z 669.715,A -85,B 0,C 180,E1 -9067.581,E2 -9067.581} C_VEL
LIN {X 0,Y 442.044,Z 672.919,A -85,B 0,C 180,E1 -9068.109,E2 -9068.109} C_VEL
LIN {X 0,Y 446.615,Z 699.659,A -85,B 0,C 180,E1 -9068.781,E2 -9068.781} C_VEL
LIN {X 0,Y 445.235,Z 810.121,A -85,B 0,C 180,E1 -9070.581,E2 -9070.581} C_VEL
LIN {X 0,Y 444.75,Z 824.539,A -85,B 0,C 180,E1 -9070.979,E2 -9070.979} C_VEL
LIN {X 0,Y 444.096,Z 838.359,A -85,B 0,C 180,E1 -9071.548,E2 -9071.548} C_VEL
LIN {X 0,Y 443.338,Z 852.4,A -85,B 0,C 180,E1 -9072.335,E2 -9072.335} C_VEL
LIN {X 0,Y 442.477,Z 865.356,A -85,B 0,C 180,E1 -9073.269,E2 -9073.269} C_VEL
LIN {X 0,Y 441.639,Z 876.947,A -85,B 0,C 180,E1 -9074.304,E2 -9074.304} C_VEL
LIN {X 0,Y 440.86,Z 887.579,A -85,B 0,C 180,E1 -9075.458,E2 -9075.458} C_VEL
LIN {X 0,Y 440.1,Z 898.305,A -85,B 0,C 180,E1 -9076.87,E2 -9076.87} C_VEL
LIN {X 0,Y 439.571,Z 906.855,A -85,B 0,C 180,E1 -9078.238,E2 -9078.238} C_VEL
LIN {X 0,Y 438.978,Z 915.201,A -85,B 0,C 180,E1 -9079.857,E2 -9079.857} C_VEL
LIN {X 0,Y 438.705,Z 921.028,A -85,B 0,C 180,E1 -9081.246,E2 -9081.246} C_VEL
LIN {X 0,Y 438.504,Z 925.813,A -85,B 0,C 180,E1 -9082.633,E2 -9082.633} C_VEL
LIN {X 0,Y 438.387,Z 930.768,A -85,B 0,C 180,E1 -9084.48,E2 -9084.48} C_VEL
LIN {X 0,Y 438.276,Z 934.211,A -85,B 0,C 180,E1 -9086.322,E2 -9086.322} C_VEL
LIN {X 0,Y 438.288,Z 936.253,A -85,B 0,C 180,E1 -9088.162,E2 -9088.162} C_VEL
LIN {X 0,Y 438.278,Z 936.937,A -85,B 0,C 180,E1 -9090,E2 -9090} C_VEL
LIN {X 0,Y 438.288,Z 936.276,A -85,B 0,C 180,E1 -9091.838,E2 -9091.838} C_VEL
LIN {X 0,Y 438.276,Z 934.258,A -85,B 0,C 180,E1 -9093.678,E2 -9093.678} C_VEL
LIN {X 0,Y 438.387,Z 930.843,A -85,B 0,C 180,E1 -9095.52,E2 -9095.52} C_VEL
LIN {X 0,Y 438.503,Z 925.927,A -85,B 0,C 180,E1 -9097.367,E2 -9097.367} C_VEL
LIN {X 0,Y 438.797,Z 919.374,A -85,B 0,C 180,E1 -9099.216,E2 -9099.216} C_VEL
LIN {X 0,Y 439.219,Z 912.096,A -85,B 0,C 180,E1 -9100.837,E2 -9100.837} C_VEL
LIN {X 0,Y 439.855,Z 903.111,A -85,B 0,C 180,E1 -9102.457,E2 -9102.457} C_VEL
LIN {X 0,Y 440.491,Z 893.693,A -85,B 0,C 180,E1 -9103.847,E2 -9103.847} C_VEL
LIN {X 0,Y 441.243,Z 883.287,A -85,B 0,C 180,E1 -9105.118,E2 -9105.118} C_VEL
LIN {X 0,Y 442.161,Z 871.833,A -85,B 0,C 180,E1 -9106.269,E2 -9106.269} C_VEL
LIN {X 0,Y 443.079,Z 859.164,A -85,B 0,C 180,E1 -9107.302,E2 -9107.302} C_VEL
LIN {X 0,Y 443.963,Z 846.047,A -85,B 0,C 180,E1 -9108.149,E2 -9108.149} C_VEL
LIN {X 0,Y 444.613,Z 833.296,A -85,B 0,C 180,E1 -9108.788,E2 -9108.788} C_VEL
LIN {X 0,Y 445.237,Z 819.27,A -85,B 0,C 180,E1 -9109.299,E2 -9109.299} C_VEL
LIN {X 0,Y 445.677,Z 804.603,A -85,B 0,C 180,E1 -9109.638,E2 -9109.638} C_VEL
LIN {X 0,Y 446.916,Z 698.809,A -85,B 0,C 180,E1 -9111.371,E2 -9111.371} C_VEL
LIN {X 0,Y 442.274,Z 672.844,A -85,B 0,C 180,E1 -9112.069,E2 -9112.069} C_VEL
LIN {X 0,Y 443.681,Z 652.773,A -85,B 0,C 180,E1 -9115.459,E2 -9115.459} C_VEL
LIN {X 0,Y 443.727,Z 649.253,A -85,B 0,C 180,E1 -9116.073,E2 -9116.073} C_VEL
LIN {X 0,Y 441.267,Z 637.72,A -85,B 0,C 180,E1 -9118.283,E2 -9118.283} C_VEL
LIN {X 0,Y 439.406,Z 629.877,A -85,B 0,C 180,E1 -9119.862,E2 -9119.862} C_VEL
LIN {X 0,Y 439.373,Z 629.874,A -85,B 0,C 180,E1 -9122.946,E2 -9122.946} C_VEL
LIN {X 0,Y 439.378,Z 629.875,A -85,B 0,C 180,E1 -9126.287,E2 -9126.287} C_VEL
LIN {X 0,Y 439.423,Z 629.869,A -85,B 0,C 180,E1 -9129.853,E2 -9129.853} C_VEL
LIN {X 0,Y 439.386,Z 629.876,A -85,B 0,C 180,E1 -9132.628,E2 -9132.628} C_VEL
LIN {X 0,Y 439.403,Z 629.874,A -85,B 0,C 180,E1 -9135.271,E2 -9135.271} C_VEL
LIN {X 0,Y 439.399,Z 629.869,A -85,B 0,C 180,E1 -9138.742,E2 -9138.742} C_VEL
LIN {X 0,Y 439.392,Z 629.871,A -85,B 0,C 180,E1 -9141.605,E2 -9141.605} C_VEL
LIN {X 0,Y 439.402,Z 629.872,A -85,B 0,C 180,E1 -9144.844,E2 -9144.844} C_VEL
LIN {X 0,Y 439.374,Z 629.862,A -85,B 0,C 180,E1 -9148.14,E2 -9148.14} C_VEL
LIN {X 0,Y 439.433,Z 629.871,A -85,B 0,C 180,E1 -9151.598,E2 -9151.598} C_VEL
LIN {X 0,Y 439.406,Z 629.872,A -85,B 0,C 180,E1 -9154.415,E2 -9154.415} C_VEL
LIN {X 0,Y 439.367,Z 629.876,A -85,B 0,C 180,E1 -9157.425,E2 -9157.425} C_VEL
LIN {X 0,Y 439.443,Z 629.866,A -85,B 0,C 180,E1 -9160.663,E2 -9160.663} C_VEL
LIN {X 0,Y 439.477,Z 629.868,A -85,B 0,C 180,E1 -9164.225,E2 -9164.225} C_VEL
LIN {X 0,Y 439.485,Z 629.866,A -85,B 0,C 180,E1 -9168.002,E2 -9168.002} C_VEL
LIN {X 0,Y 439.55,Z 629.851,A -85,B 0,C 180,E1 -9171.727,E2 -9171.727} C_VEL
LIN {X 0,Y 439.621,Z 629.845,A -85,B 0,C 180,E1 -9174.496,E2 -9174.496} C_VEL
LIN {X 0,Y 439.635,Z 629.849,A -85,B 0,C 180,E1 -9178.168,E2 -9178.168} C_VEL
LIN {X 0,Y 439.764,Z 629.83,A -85,B 0,C 180,E1 -9180,E2 -9180} C_VEL
LIN {X 0,Y 439.642,Z 629.846,A -85,B 0,C 180,E1 -9182.749,E2 -9182.749} C_VEL
LIN {X 0,Y 439.613,Z 629.847,A -85,B 0,C 180,E1 -9186.426,E2 -9186.426} C_VEL
LIN {X 0,Y 439.5,Z 629.858,A -85,B 0,C 180,E1 -9189.202,E2 -9189.202} C_VEL
LIN {X 0,Y 439.468,Z 629.867,A -85,B 0,C 180,E1 -9192.938,E2 -9192.938} C_VEL
LIN {X 0,Y 439.448,Z 629.867,A -85,B 0,C 180,E1 -9196.349,E2 -9196.349} C_VEL
LIN {X 0,Y 439.404,Z 629.868,A -85,B 0,C 180,E1 -9199.627,E2 -9199.627} C_VEL
LIN {X 0,Y 439.367,Z 629.882,A -85,B 0,C 180,E1 -9202.576,E2 -9202.576} C_VEL
LIN {X 0,Y 439.384,Z 629.875,A -85,B 0,C 180,E1 -9205.587,E2 -9205.587} C_VEL
LIN {X 0,Y 439.402,Z 629.862,A -85,B 0,C 180,E1 -9208.675,E2 -9208.675} C_VEL
LIN {X 0,Y 439.371,Z 629.876,A -85,B 0,C 180,E1 -9212.03,E2 -9212.03} C_VEL
LIN {X 0,Y 439.394,Z 629.877,A -85,B 0,C 180,E1 -9215.34,E2 -9215.34} C_VEL
LIN {X 0,Y 439.37,Z 629.88,A -85,B 0,C 180,E1 -9218.597,E2 -9218.597} C_VEL
LIN {X 0,Y 439.369,Z 629.873,A -85,B 0,C 180,E1 -9221.254,E2 -9221.254} C_VEL
LIN {X 0,Y 439.4,Z 629.876,A -85,B 0,C 180,E1 -9224.73,E2 -9224.73} C_VEL
LIN {X 0,Y 439.353,Z 629.883,A -85,B 0,C 180,E1 -9227.791,E2 -9227.791} C_VEL
LIN {X 0,Y 439.361,Z 629.881,A -85,B 0,C 180,E1 -9230.22,E2 -9230.22} C_VEL
LIN {X 0,Y 439.376,Z 629.878,A -85,B 0,C 180,E1 -9233.713,E2 -9233.713} C_VEL
LIN {X 0,Y 439.373,Z 629.87,A -85,B 0,C 180,E1 -9237.054,E2 -9237.054} C_VEL
LIN {X 0,Y 439.419,Z 629.976,A -85,B 0,C 180,E1 -9240.116,E2 -9240.116} C_VEL
LIN {X 0,Y 442.043,Z 642.503,A -85,B 0,C 180,E1 -9242.965,E2 -9242.965} C_VEL
LIN {X 0,Y 444.49,Z 650.821,A -85,B 0,C 180,E1 -9243.256,E2 -9243.256} C_VEL
LIN {X 0,Y 447.27,Z 663.431,A -85,B 0,C 180,E1 -9243.625,E2 -9243.625} C_VEL
LIN {X 0,Y 445.877,Z 778.33,A -85,B 0,C 180,E1 -9245.528,E2 -9245.528} C_VEL
LIN {X 0,Y 445.393,Z 792.703,A -85,B 0,C 180,E1 -9245.939,E2 -9245.939} C_VEL
LIN {X 0,Y 444.706,Z 806.144,A -85,B 0,C 180,E1 -9246.501,E2 -9246.501} C_VEL
LIN {X 0,Y 444.068,Z 818.386,A -85,B 0,C 180,E1 -9247.186,E2 -9247.186} C_VEL
LIN {X 0,Y 443.762,Z 823.561,A -85,B 0,C 180,E1 -9247.527,E2 -9247.527} C_VEL
LIN {X 0,Y 442.813,Z 828.76,A -85,B 0,C 180,E1 -9247.869,E2 -9247.869} C_VEL
LIN {X 0,Y 439.505,Z 837.05,A -85,B 0,C 180,E1 -9248.431,E2 -9248.431} C_VEL
LIN {X 0,Y 436.147,Z 844.998,A -85,B 0,C 180,E1 -9249.073,E2 -9249.073} C_VEL
LIN {X 0,Y 435.132,Z 849.583,A -85,B 0,C 180,E1 -9249.538,E2 -9249.538} C_VEL
LIN {X 0,Y 434.215,Z 860.386,A -85,B 0,C 180,E1 -9250.867,E2 -9250.867} C_VEL
LIN {X 0,Y 433.401,Z 869.945,A -85,B 0,C 180,E1 -9252.299,E2 -9252.299} C_VEL
LIN {X 0,Y 432.704,Z 879.012,A -85,B 0,C 180,E1 -9253.972,E2 -9253.972} C_VEL
LIN {X 0,Y 432.143,Z 885.369,A -85,B 0,C 180,E1 -9255.4,E2 -9255.4} C_VEL
LIN {X 0,Y 431.835,Z 890.564,A -85,B 0,C 180,E1 -9256.83,E2 -9256.83} C_VEL
LIN {X 0,Y 431.512,Z 896.024,A -85,B 0,C 180,E1 -9258.729,E2 -9258.729} C_VEL
LIN {X 0,Y 431.301,Z 899.882,A -85,B 0,C 180,E1 -9260.622,E2 -9260.622} C_VEL
LIN {X 0,Y 431.26,Z 902.305,A -85,B 0,C 180,E1 -9262.509,E2 -9262.509} C_VEL
LIN {X 0,Y 431.234,Z 903.384,A -85,B 0,C 180,E1 -9264.388,E2 -9264.388} C_VEL
LIN {X 0,Y 431.185,Z 903.15,A -85,B 0,C 180,E1 -9266.262,E2 -9266.262} C_VEL
LIN {X 0,Y 431.284,Z 902.537,A -85,B 0,C 180,E1 -9267.198,E2 -9267.198} C_VEL
LIN {X 0,Y 431.251,Z 900.328,A -85,B 0,C 180,E1 -9269.066,E2 -9269.066} C_VEL
LIN {X 0,Y 431.353,Z 896.745,A -85,B 0,C 180,E1 -9270.934,E2 -9270.934} C_VEL
LIN {X 0,Y 431.655,Z 891.682,A -85,B 0,C 180,E1 -9272.8,E2 -9272.8} C_VEL
LIN {X 0,Y 432.075,Z 886.769,A -85,B 0,C 180,E1 -9274.198,E2 -9274.198} C_VEL
LIN {X 0,Y 432.62,Z 879.747,A -85,B 0,C 180,E1 -9275.828,E2 -9275.828} C_VEL
LIN {X 0,Y 433.074,Z 872.423,A -85,B 0,C 180,E1 -9277.225,E2 -9277.225} C_VEL
LIN {X 0,Y 433.684,Z 863.789,A -85,B 0,C 180,E1 -9278.598,E2 -9278.598} C_VEL
LIN {X 0,Y 434.499,Z 854.893,A -85,B 0,C 180,E1 -9279.778,E2 -9279.778} C_VEL
LIN {X 0,Y 435.406,Z 843.341,A -85,B 0,C 180,E1 -9281.051,E2 -9281.051} C_VEL
LIN {X 0,Y 436.186,Z 831.792,A -85,B 0,C 180,E1 -9282.091,E2 -9282.091} C_VEL
LIN {X 0,Y 437.044,Z 819.073,A -85,B 0,C 180,E1 -9283.011,E2 -9283.011} C_VEL
LIN {X 0,Y 437.773,Z 805.858,A -85,B 0,C 180,E1 -9283.757,E2 -9283.757} C_VEL
LIN {X 0,Y 438.269,Z 792.237,A -85,B 0,C 180,E1 -9284.333,E2 -9284.333} C_VEL
LIN {X 0,Y 438.648,Z 778.086,A -85,B 0,C 180,E1 -9284.735,E2 -9284.735} C_VEL
LIN {X 0,Y 440.167,Z 665.154,A -85,B 0,C 180,E1 -9286.604,E2 -9286.604} C_VEL
LIN {X 0,Y 438.777,Z 657.884,A -85,B 0,C 180,E1 -9286.797,E2 -9286.797} C_VEL
LIN {X 0,Y 435.668,Z 645.271,A -85,B 0,C 180,E1 -9287.168,E2 -9287.168} C_VEL
LIN {X 0,Y 434.796,Z 642.598,A -85,B 0,C 180,E1 -9287.279,E2 -9287.279} C_VEL
LIN {X 0,Y 432.395,Z 630.753,A -85,B 0,C 180,E1 -9289.958,E2 -9289.958} C_VEL
LIN {X 0,Y 432.313,Z 630.762,A -85,B 0,C 180,E1 -9292.965,E2 -9292.965} C_VEL
LIN {X 0,Y 432.309,Z 630.76,A -85,B 0,C 180,E1 -9296.036,E2 -9296.036} C_VEL
LIN {X 0,Y 432.324,Z 630.758,A -85,B 0,C 180,E1 -9299.189,E2 -9299.189} C_VEL
LIN {X 0,Y 432.308,Z 630.761,A -85,B 0,C 180,E1 -9302.444,E2 -9302.444} C_VEL
LIN {X 0,Y 432.335,Z 630.753,A -85,B 0,C 180,E1 -9305.818,E2 -9305.818} C_VEL
LIN {X 0,Y 432.303,Z 630.75,A -85,B 0,C 180,E1 -9309.348,E2 -9309.348} C_VEL
LIN {X 0,Y 432.306,Z 630.757,A -85,B 0,C 180,E1 -9311.801,E2 -9311.801} C_VEL
LIN {X 0,Y 432.336,Z 630.751,A -85,B 0,C 180,E1 -9314.347,E2 -9314.347} C_VEL
LIN {X 0,Y 432.305,Z 630.76,A -85,B 0,C 180,E1 -9317.018,E2 -9317.018} C_VEL
LIN {X 0,Y 432.291,Z 630.757,A -85,B 0,C 180,E1 -9319.828,E2 -9319.828} C_VEL
LIN {X 0,Y 432.304,Z 630.744,A -85,B 0,C 180,E1 -9323.021,E2 -9323.021} C_VEL
LIN {X 0,Y 432.361,Z 630.749,A -85,B 0,C 180,E1 -9325.997,E2 -9325.997} C_VEL
LIN {X 0,Y 432.349,Z 630.748,A -85,B 0,C 180,E1 -9329.49,E2 -9329.49} C_VEL
LIN {X 0,Y 432.338,Z 630.754,A -85,B 0,C 180,E1 -9331.873,E2 -9331.873} C_VEL
LIN {X 0,Y 432.355,Z 630.746,A -85,B 0,C 180,E1 -9335.546,E2 -9335.546} C_VEL
LIN {X 0,Y 432.354,Z 630.753,A -85,B 0,C 180,E1 -9339.046,E2 -9339.046} C_VEL
LIN {X 0,Y 432.364,Z 630.74,A -85,B 0,C 180,E1 -9342.01,E2 -9342.01} C_VEL
LIN {X 0,Y 432.398,Z 630.744,A -85,B 0,C 180,E1 -9344.926,E2 -9344.926} C_VEL
LIN {X 0,Y 432.462,Z 630.736,A -85,B 0,C 180,E1 -9347.803,E2 -9347.803} C_VEL
LIN {X 0,Y 432.467,Z 630.737,A -85,B 0,C 180,E1 -9351.59,E2 -9351.59} C_VEL
LIN {X 0,Y 432.582,Z 630.721,A -85,B 0,C 180,E1 -9354.406,E2 -9354.406} C_VEL
LIN {X 0,Y 432.605,Z 630.722,A -85,B 0,C 180,E1 -9358.138,E2 -9358.138} C_VEL
LIN {X 0,Y 432.733,Z 630.703,A -85,B 0,C 180,E1 -9360,E2 -9360} C_VEL
LIN {X 0,Y 432.594,Z 630.72,A -85,B 0,C 180,E1 -9362.793,E2 -9362.793} C_VEL
LIN {X 0,Y 432.589,Z 630.723,A -85,B 0,C 180,E1 -9365.594,E2 -9365.594} C_VEL
LIN {X 0,Y 432.485,Z 630.736,A -85,B 0,C 180,E1 -9368.41,E2 -9368.41} C_VEL
LIN {X 0,Y 432.462,Z 630.742,A -85,B 0,C 180,E1 -9372.196,E2 -9372.196} C_VEL
LIN {X 0,Y 432.446,Z 630.741,A -85,B 0,C 180,E1 -9376.038,E2 -9376.038} C_VEL
LIN {X 0,Y 432.389,Z 630.743,A -85,B 0,C 180,E1 -9379.485,E2 -9379.485} C_VEL
LIN {X 0,Y 432.32,Z 630.751,A -85,B 0,C 180,E1 -9382.964,E2 -9382.964} C_VEL
LIN {X 0,Y 432.363,Z 630.753,A -85,B 0,C 180,E1 -9386.032,E2 -9386.032} C_VEL
LIN {X 0,Y 432.345,Z 630.751,A -85,B 0,C 180,E1 -9389.187,E2 -9389.187} C_VEL
LIN {X 0,Y 432.325,Z 630.76,A -85,B 0,C 180,E1 -9392.443,E2 -9392.443} C_VEL
LIN {X 0,Y 432.346,Z 630.752,A -85,B 0,C 180,E1 -9395.632,E2 -9395.632} C_VEL
LIN {X 0,Y 432.359,Z 630.752,A -85,B 0,C 180,E1 -9398.717,E2 -9398.717} C_VEL
LIN {X 0,Y 432.367,Z 630.749,A -85,B 0,C 180,E1 -9401.793,E2 -9401.793} C_VEL
LIN {X 0,Y 432.335,Z 630.756,A -85,B 0,C 180,E1 -9404.347,E2 -9404.347} C_VEL
LIN {X 0,Y 432.326,Z 630.754,A -85,B 0,C 180,E1 -9407.015,E2 -9407.015} C_VEL
LIN {X 0,Y 432.343,Z 630.753,A -85,B 0,C 180,E1 -9409.819,E2 -9409.819} C_VEL
LIN {X 0,Y 432.318,Z 630.76,A -85,B 0,C 180,E1 -9413.023,E2 -9413.023} C_VEL
LIN {X 0,Y 432.361,Z 630.753,A -85,B 0,C 180,E1 -9415.996,E2 -9415.996} C_VEL
LIN {X 0,Y 432.349,Z 630.753,A -85,B 0,C 180,E1 -9419.489,E2 -9419.489} C_VEL
LIN {X 0,Y 432.386,Z 630.831,A -85,B 0,C 180,E1 -9420.281,E2 -9420.281} C_VEL
LIN {X 0,Y 435.375,Z 644.094,A -85,B 0,C 180,E1 -9422.832,E2 -9422.832} C_VEL
LIN {X 0,Y 436.578,Z 650.285,A -85,B 0,C 180,E1 -9423.981,E2 -9423.981} C_VEL
LIN {X 0,Y 435.569,Z 667.367,A -85,B 0,C 180,E1 -9426.883,E2 -9426.883} C_VEL
LIN {X 0,Y 435.167,Z 672.699,A -85,B 0,C 180,E1 -9427.777,E2 -9427.777} C_VEL
LIN {X 0,Y 439.912,Z 699.832,A -85,B 0,C 180,E1 -9428.472,E2 -9428.472} C_VEL
LIN {X 0,Y 438.478,Z 810.282,A -85,B 0,C 180,E1 -9430.3,E2 -9430.3} C_VEL
LIN {X 0,Y 437.991,Z 824.502,A -85,B 0,C 180,E1 -9430.704,E2 -9430.704} C_VEL
LIN {X 0,Y 437.326,Z 837.693,A -85,B 0,C 180,E1 -9431.252,E2 -9431.252} C_VEL
LIN {X 0,Y 436.659,Z 850.341,A -85,B 0,C 180,E1 -9431.955,E2 -9431.955} C_VEL
LIN {X 0,Y 435.749,Z 863.405,A -85,B 0,C 180,E1 -9432.882,E2 -9432.882} C_VEL
LIN {X 0,Y 434.793,Z 875.29,A -85,B 0,C 180,E1 -9433.93,E2 -9433.93} C_VEL
LIN {X 0,Y 433.926,Z 887.147,A -85,B 0,C 180,E1 -9435.221,E2 -9435.221} C_VEL
LIN {X 0,Y 433.144,Z 897.738,A -85,B 0,C 180,E1 -9436.631,E2 -9436.631} C_VEL
LIN {X 0,Y 432.537,Z 906.476,A -85,B 0,C 180,E1 -9438.044,E2 -9438.044} C_VEL
LIN {X 0,Y 431.938,Z 914.85,A -85,B 0,C 180,E1 -9439.69,E2 -9439.69} C_VEL
LIN {X 0,Y 431.63,Z 920.689,A -85,B 0,C 180,E1 -9441.101,E2 -9441.101} C_VEL
LIN {X 0,Y 431.41,Z 925.49,A -85,B 0,C 180,E1 -9442.511,E2 -9442.511} C_VEL
LIN {X 0,Y 431.355,Z 928.703,A -85,B 0,C 180,E1 -9443.649,E2 -9443.649} C_VEL
LIN {X 0,Y 431.251,Z 932.368,A -85,B 0,C 180,E1 -9445.326,E2 -9445.326} C_VEL
LIN {X 0,Y 431.238,Z 935.114,A -85,B 0,C 180,E1 -9447.197,E2 -9447.197} C_VEL
LIN {X 0,Y 431.189,Z 936.484,A -85,B 0,C 180,E1 -9449.066,E2 -9449.066} C_VEL
LIN {X 0,Y 431.189,Z 936.506,A -85,B 0,C 180,E1 -9450.934,E2 -9450.934} C_VEL
LIN {X 0,Y 431.223,Z 935.183,A -85,B 0,C 180,E1 -9452.802,E2 -9452.802} C_VEL
LIN {X 0,Y 431.251,Z 932.486,A -85,B 0,C 180,E1 -9454.674,E2 -9454.674} C_VEL
LIN {X 0,Y 431.372,Z 928.348,A -85,B 0,C 180,E1 -9456.548,E2 -9456.548} C_VEL
LIN {X 0,Y 431.569,Z 922.648,A -85,B 0,C 180,E1 -9458.428,E2 -9458.428} C_VEL
LIN {X 0,Y 431.899,Z 916.235,A -85,B 0,C 180,E1 -9460.074,E2 -9460.074} C_VEL
LIN {X 0,Y 432.49,Z 908.279,A -85,B 0,C 180,E1 -9461.72,E2 -9461.72} C_VEL
LIN {X 0,Y 433.124,Z 899.535,A -85,B 0,C 180,E1 -9463.2,E2 -9463.2} C_VEL
LIN {X 0,Y 433.819,Z 889.989,A -85,B 0,C 180,E1 -9464.543,E2 -9464.543} C_VEL
LIN {X 0,Y 434.717,Z 878.905,A -85,B 0,C 180,E1 -9465.832,E2 -9465.832} C_VEL
LIN {X 0,Y 435.769,Z 866.529,A -85,B 0,C 180,E1 -9466.997,E2 -9466.997} C_VEL
LIN {X 0,Y 436.654,Z 854.115,A -85,B 0,C 180,E1 -9467.94,E2 -9467.94} C_VEL
LIN {X 0,Y 437.497,Z 840.691,A -85,B 0,C 180,E1 -9468.74,E2 -9468.74} C_VEL
LIN {X 0,Y 438.288,Z 826.424,A -85,B 0,C 180,E1 -9469.374,E2 -9469.374} C_VEL
LIN {X 0,Y 438.895,Z 812.313,A -85,B 0,C 180,E1 -9469.802,E2 -9469.802} C_VEL
LIN {X 0,Y 439.324,Z 784.348,A -85,B 0,C 180,E1 -9470.3,E2 -9470.3} C_VEL
LIN {X 0,Y 440.398,Z 699.885,A -85,B 0,C 180,E1 -9471.703,E2 -9471.703} C_VEL
LIN {X 0,Y 435.479,Z 672.515,A -85,B 0,C 180,E1 -9472.466,E2 -9472.466} C_VEL
LIN {X 0,Y 436.898,Z 653.46,A -85,B 0,C 180,E1 -9475.742,E2 -9475.742} C_VEL
LIN {X 0,Y 436.562,Z 649.146,A -85,B 0,C 180,E1 -9476.534,E2 -9476.534} C_VEL
LIN {X 0,Y 433.705,Z 636.198,A -85,B 0,C 180,E1 -9479.087,E2 -9479.087} C_VEL
LIN {X 0,Y 432.337,Z 630.756,A -85,B 0,C 180,E1 -9480.227,E2 -9480.227} C_VEL
LIN {X 0,Y 432.34,Z 630.751,A -85,B 0,C 180,E1 -9483.552,E2 -9483.552} C_VEL
LIN {X 0,Y 432.341,Z 630.753,A -85,B 0,C 180,E1 -9485.817,E2 -9485.817} C_VEL
LIN {X 0,Y 432.363,Z 630.755,A -85,B 0,C 180,E1 -9489.341,E2 -9489.341} C_VEL
LIN {X 0,Y 432.366,Z 630.754,A -85,B 0,C 180,E1 -9491.793,E2 -9491.793} C_VEL
LIN {X 0,Y 432.341,Z 630.749,A -85,B 0,C 180,E1 -9494.346,E2 -9494.346} C_VEL
LIN {X 0,Y 432.321,Z 630.756,A -85,B 0,C 180,E1 -9497.016,E2 -9497.016} C_VEL
LIN {X 0,Y 432.357,Z 630.755,A -85,B 0,C 180,E1 -9499.817,E2 -9499.817} C_VEL
LIN {X 0,Y 432.317,Z 630.744,A -85,B 0,C 180,E1 -9503.023,E2 -9503.023} C_VEL
LIN {X 0,Y 432.36,Z 630.751,A -85,B 0,C 180,E1 -9505.996,E2 -9505.996} C_VEL
LIN {X 0,Y 432.348,Z 630.739,A -85,B 0,C 180,E1 -9509.49,E2 -9509.49} C_VEL
LIN {X 0,Y 432.393,Z 630.744,A -85,B 0,C 180,E1 -9512.929,E2 -9512.929} C_VEL
LIN {X 0,Y 432.373,Z 630.751,A -85,B 0,C 180,E1 -9516.024,E2 -9516.024} C_VEL
LIN {X 0,Y 432.352,Z 630.75,A -85,B 0,C 180,E1 -9519.046,E2 -9519.046} C_VEL
LIN {X 0,Y 432.381,Z 630.748,A -85,B 0,C 180,E1 -9522.011,E2 -9522.011} C_VEL
LIN {X 0,Y 432.403,Z 630.743,A -85,B 0,C 180,E1 -9524.927,E2 -9524.927} C_VEL
LIN {X 0,Y 432.461,Z 630.739,A -85,B 0,C 180,E1 -9527.804,E2 -9527.804} C_VEL
LIN {X 0,Y 432.494,Z 630.729,A -85,B 0,C 180,E1 -9531.591,E2 -9531.591} C_VEL
LIN {X 0,Y 432.597,Z 630.721,A -85,B 0,C 180,E1 -9534.406,E2 -9534.406} C_VEL
LIN {X 0,Y 432.605,Z 630.724,A -85,B 0,C 180,E1 -9538.138,E2 -9538.138} C_VEL
LIN {X 0,Y 432.734,Z 630.705,A -85,B 0,C 180,E1 -9540,E2 -9540} C_VEL
LIN {X 0,Y 432.594,Z 630.724,A -85,B 0,C 180,E1 -9542.794,E2 -9542.794} C_VEL
LIN {X 0,Y 432.566,Z 630.726,A -85,B 0,C 180,E1 -9546.531,E2 -9546.531} C_VEL
LIN {X 0,Y 432.443,Z 630.737,A -85,B 0,C 180,E1 -9549.353,E2 -9549.353} C_VEL
LIN {X 0,Y 432.433,Z 630.745,A -85,B 0,C 180,E1 -9552.804,E2 -9552.804} C_VEL
LIN {X 0,Y 432.414,Z 630.745,A -85,B 0,C 180,E1 -9556.479,E2 -9556.479} C_VEL
LIN {X 0,Y 432.341,Z 630.748,A -85,B 0,C 180,E1 -9559.961,E2 -9559.961} C_VEL
LIN {X 0,Y 432.321,Z 630.755,A -85,B 0,C 180,E1 -9562.965,E2 -9562.965} C_VEL
LIN {X 0,Y 432.343,Z 630.757,A -85,B 0,C 180,E1 -9565.002,E2 -9565.002} C_VEL
LIN {X 0,Y 432.349,Z 630.744,A -85,B 0,C 180,E1 -9568.126,E2 -9568.126} C_VEL
LIN {X 0,Y 432.322,Z 630.757,A -85,B 0,C 180,E1 -9571.346,E2 -9571.346} C_VEL
LIN {X 0,Y 432.34,Z 630.753,A -85,B 0,C 180,E1 -9574.678,E2 -9574.678} C_VEL
LIN {X 0,Y 432.334,Z 630.754,A -85,B 0,C 180,E1 -9578.151,E2 -9578.151} C_VEL
LIN {X 0,Y 432.313,Z 630.755,A -85,B 0,C 180,E1 -9581.599,E2 -9581.599} C_VEL
LIN {X 0,Y 432.336,Z 630.754,A -85,B 0,C 180,E1 -9584.348,E2 -9584.348} C_VEL
LIN {X 0,Y 432.306,Z 630.762,A -85,B 0,C 180,E1 -9587.018,E2 -9587.018} C_VEL
LIN {X 0,Y 432.31,Z 630.761,A -85,B 0,C 180,E1 -9589.825,E2 -9589.825} C_VEL
LIN {X 0,Y 432.309,Z 630.762,A -85,B 0,C 180,E1 -9593.022,E2 -9593.022} C_VEL
LIN {X 0,Y 432.336,Z 630.753,A -85,B 0,C 180,E1 -9596.002,E2 -9596.002} C_VEL
LIN {X 0,Y 432.344,Z 630.756,A -85,B 0,C 180,E1 -9599.491,E2 -9599.491} C_VEL
LIN {X 0,Y 432.387,Z 630.961,A -85,B 0,C 180,E1 -9599.811,E2 -9599.811} C_VEL
LIN {X 0,Y 434.811,Z 642.291,A -85,B 0,C 180,E1 -9602.441,E2 -9602.441} C_VEL
LIN {X 0,Y 434.922,Z 642.869,A -85,B 0,C 180,E1 -9602.565,E2 -9602.565} C_VEL
LIN {X 0,Y 437.688,Z 650.963,A -85,B 0,C 180,E1 -9602.871,E2 -9602.871} C_VEL
LIN {X 0,Y 440.757,Z 664.89,A -85,B 0,C 180,E1 -9603.29,E2 -9603.29} C_VEL
LIN {X 0,Y 439.274,Z 778.546,A -85,B 0,C 180,E1 -9605.198,E2 -9605.198} C_VEL
LIN {X 0,Y 438.776,Z 792.538,A -85,B 0,C 180,E1 -9605.599,E2 -9605.599} C_VEL
LIN {X 0,Y 438.135,Z 805.237,A -85,B 0,C 180,E1 -9606.127,E2 -9606.127} C_VEL
LIN {X 0,Y 437.441,Z 817.73,A -85,B 0,C 180,E1 -9606.82,E2 -9606.82} C_VEL
LIN {X 0,Y 436.514,Z 831.01,A -85,B 0,C 180,E1 -9607.768,E2 -9607.768} C_VEL
LIN {X 0,Y 435.641,Z 842.969,A -85,B 0,C 180,E1 -9608.841,E2 -9608.841} C_VEL
LIN {X 0,Y 435.132,Z 849.583,A -85,B 0,C 180,E1 -9609.538,E2 -9609.538} C_VEL
LIN {X 0,Y 434.117,Z 854.08,A -85,B 0,C 180,E1 -9610.027,E2 -9610.027} C_VEL
LIN {X 0,Y 430.734,Z 861.219,A -85,B 0,C 180,E1 -9610.824,E2 -9610.824} C_VEL
LIN {X 0,Y 427.36,Z 867.857,A -85,B 0,C 180,E1 -9611.697,E2 -9611.697} C_VEL
LIN {X 0,Y 426.371,Z 871.569,A -85,B 0,C 180,E1 -9612.299,E2 -9612.299} C_VEL
LIN {X 0,Y 425.656,Z 880.116,A -85,B 0,C 180,E1 -9613.945,E2 -9613.945} C_VEL
LIN {X 0,Y 425.037,Z 887.229,A -85,B 0,C 180,E1 -9615.639,E2 -9615.639} C_VEL
LIN {X 0,Y 424.7,Z 892.165,A -85,B 0,C 180,E1 -9617.091,E2 -9617.091} C_VEL
LIN {X 0,Y 424.403,Z 897.233,A -85,B 0,C 180,E1 -9619.022,E2 -9619.022} C_VEL
LIN {X 0,Y 424.222,Z 900.06,A -85,B 0,C 180,E1 -9620.464,E2 -9620.464} C_VEL
LIN {X 0,Y 424.175,Z 902.526,A -85,B 0,C 180,E1 -9622.383,E2 -9622.383} C_VEL
LIN {X 0,Y 424.145,Z 903.647,A -85,B 0,C 180,E1 -9624.294,E2 -9624.294} C_VEL
LIN {X 0,Y 424.092,Z 903.455,A -85,B 0,C 180,E1 -9626.199,E2 -9626.199} C_VEL
LIN {X 0,Y 424.179,Z 901.946,A -85,B 0,C 180,E1 -9628.101,E2 -9628.101} C_VEL
LIN {X 0,Y 424.197,Z 899.103,A -85,B 0,C 180,E1 -9630,E2 -9630} C_VEL
LIN {X 0,Y 424.388,Z 894.843,A -85,B 0,C 180,E1 -9631.898,E2 -9631.898} C_VEL
LIN {X 0,Y 424.855,Z 889.03,A -85,B 0,C 180,E1 -9633.794,E2 -9633.794} C_VEL
LIN {X 0,Y 425.369,Z 882.492,A -85,B 0,C 180,E1 -9635.452,E2 -9635.452} C_VEL
LIN {X 0,Y 426.027,Z 874.373,A -85,B 0,C 180,E1 -9637.107,E2 -9637.107} C_VEL
LIN {X 0,Y 426.557,Z 865.925,A -85,B 0,C 180,E1 -9638.528,E2 -9638.528} C_VEL
LIN {X 0,Y 427.569,Z 855.659,A -85,B 0,C 180,E1 -9639.939,E2 -9639.939} C_VEL
LIN {X 0,Y 428.505,Z 844.206,A -85,B 0,C 180,E1 -9641.231,E2 -9641.231} C_VEL
LIN {X 0,Y 429.319,Z 832.779,A -85,B 0,C 180,E1 -9642.287,E2 -9642.287} C_VEL
LIN {X 0,Y 430.218,Z 820.225,A -85,B 0,C 180,E1 -9643.221,E2 -9643.221} C_VEL
LIN {X 0,Y 430.936,Z 807.261,A -85,B 0,C 180,E1 -9643.979,E2 -9643.979} C_VEL
LIN {X 0,Y 431.496,Z 793.282,A -85,B 0,C 180,E1 -9644.593,E2 -9644.593} C_VEL
LIN {X 0,Y 431.913,Z 779.64,A -85,B 0,C 180,E1 -9645,E2 -9645} C_VEL
LIN {X 0,Y 433.456,Z 665.043,A -85,B 0,C 180,E1 -9646.937,E2 -9646.937} C_VEL
LIN {X 0,Y 429.422,Z 648.029,A -85,B 0,C 180,E1 -9647.439,E2 -9647.439} C_VEL
LIN {X 0,Y 427.642,Z 642.901,A -85,B 0,C 180,E1 -9647.637,E2 -9647.637} C_VEL
LIN {X 0,Y 425.334,Z 631.633,A -85,B 0,C 180,E1 -9650.218,E2 -9650.218} C_VEL
LIN {X 0,Y 425.272,Z 631.637,A -85,B 0,C 180,E1 -9653.367,E2 -9653.367} C_VEL
LIN {X 0,Y 425.264,Z 631.638,A -85,B 0,C 180,E1 -9656.501,E2 -9656.501} C_VEL
LIN {X 0,Y 425.281,Z 631.633,A -85,B 0,C 180,E1 -9659.721,E2 -9659.721} C_VEL
LIN {X 0,Y 425.263,Z 631.64,A -85,B 0,C 180,E1 -9663.05,E2 -9663.05} C_VEL
LIN {X 0,Y 425.279,Z 631.632,A -85,B 0,C 180,E1 -9665.927,E2 -9665.927} C_VEL
LIN {X 0,Y 425.262,Z 631.63,A -85,B 0,C 180,E1 -9669.037,E2 -9669.037} C_VEL
LIN {X 0,Y 425.259,Z 631.638,A -85,B 0,C 180,E1 -9672.655,E2 -9672.655} C_VEL
LIN {X 0,Y 425.288,Z 631.635,A -85,B 0,C 180,E1 -9675.283,E2 -9675.283} C_VEL
LIN {X 0,Y 425.25,Z 631.637,A -85,B 0,C 180,E1 -9678.618,E2 -9678.618} C_VEL
LIN {X 0,Y 425.28,Z 631.627,A -85,B 0,C 180,E1 -9681.099,E2 -9681.099} C_VEL
LIN {X 0,Y 425.3,Z 631.622,A -85,B 0,C 180,E1 -9684.664,E2 -9684.664} C_VEL
LIN {X 0,Y 425.267,Z 631.632,A -85,B 0,C 180,E1 -9688.073,E2 -9688.073} C_VEL
LIN {X 0,Y 425.312,Z 631.63,A -85,B 0,C 180,E1 -9691.366,E2 -9691.366} C_VEL
LIN {X 0,Y 425.264,Z 631.631,A -85,B 0,C 180,E1 -9694.552,E2 -9694.552} C_VEL
LIN {X 0,Y 425.295,Z 631.633,A -85,B 0,C 180,E1 -9697.729,E2 -9697.729} C_VEL
LIN {X 0,Y 425.364,Z 631.619,A -85,B 0,C 180,E1 -9700.704,E2 -9700.704} C_VEL
LIN {X 0,Y 425.391,Z 631.617,A -85,B 0,C 180,E1 -9703.688,E2 -9703.688} C_VEL
LIN {X 0,Y 425.415,Z 631.616,A -85,B 0,C 180,E1 -9707.598,E2 -9707.598} C_VEL
LIN {X 0,Y 425.411,Z 631.614,A -85,B 0,C 180,E1 -9711.449,E2 -9711.449} C_VEL
LIN {X 0,Y 425.535,Z 631.599,A -85,B 0,C 180,E1 -9714.313,E2 -9714.313} C_VEL
LIN {X 0,Y 425.574,Z 631.598,A -85,B 0,C 180,E1 -9718.107,E2 -9718.107} C_VEL
LIN {X 0,Y 425.702,Z 631.579,A -85,B 0,C 180,E1 -9720,E2 -9720} C_VEL
LIN {X 0,Y 425.547,Z 631.598,A -85,B 0,C 180,E1 -9722.84,E2 -9722.84} C_VEL
LIN {X 0,Y 425.544,Z 631.601,A -85,B 0,C 180,E1 -9725.687,E2 -9725.687} C_VEL
LIN {X 0,Y 425.439,Z 631.613,A -85,B 0,C 180,E1 -9728.55,E2 -9728.55} C_VEL
LIN {X 0,Y 425.415,Z 631.617,A -85,B 0,C 180,E1 -9732.401,E2 -9732.401} C_VEL
LIN {X 0,Y 425.402,Z 631.62,A -85,B 0,C 180,E1 -9736.311,E2 -9736.311} C_VEL
LIN {X 0,Y 425.331,Z 631.624,A -85,B 0,C 180,E1 -9739.636,E2 -9739.636} C_VEL
LIN {X 0,Y 425.29,Z 631.632,A -85,B 0,C 180,E1 -9742.338,E2 -9742.338} C_VEL
LIN {X 0,Y 425.292,Z 631.629,A -85,B 0,C 180,E1 -9745.445,E2 -9745.445} C_VEL
LIN {X 0,Y 425.35,Z 631.62,A -85,B 0,C 180,E1 -9747.557,E2 -9747.557} C_VEL
LIN {X 0,Y 425.289,Z 631.631,A -85,B 0,C 180,E1 -9750.816,E2 -9750.816} C_VEL
LIN {X 0,Y 425.313,Z 631.631,A -85,B 0,C 180,E1 -9754.288,E2 -9754.288} C_VEL
LIN {X 0,Y 425.289,Z 631.631,A -85,B 0,C 180,E1 -9757.693,E2 -9757.693} C_VEL
LIN {X 0,Y 425.301,Z 631.636,A -85,B 0,C 180,E1 -9760.523,E2 -9760.523} C_VEL
LIN {X 0,Y 425.259,Z 631.634,A -85,B 0,C 180,E1 -9763.351,E2 -9763.351} C_VEL
LIN {X 0,Y 425.265,Z 631.633,A -85,B 0,C 180,E1 -9766.648,E2 -9766.648} C_VEL
LIN {X 0,Y 425.296,Z 631.631,A -85,B 0,C 180,E1 -9769.874,E2 -9769.874} C_VEL
LIN {X 0,Y 425.286,Z 631.637,A -85,B 0,C 180,E1 -9772.487,E2 -9772.487} C_VEL
LIN {X 0,Y 425.309,Z 631.631,A -85,B 0,C 180,E1 -9775.817,E2 -9775.817} C_VEL
LIN {X 0,Y 425.292,Z 631.629,A -85,B 0,C 180,E1 -9779.239,E2 -9779.239} C_VEL
LIN {X 0,Y 425.319,Z 631.674,A -85,B 0,C 180,E1 -9779.975,E2 -9779.975} C_VEL
LIN {X 0,Y 428.431,Z 645.355,A -85,B 0,C 180,E1 -9782.657,E2 -9782.657} C_VEL
LIN {X 0,Y 429.628,Z 651.323,A -85,B 0,C 180,E1 -9783.789,E2 -9783.789} C_VEL
LIN {X 0,Y 429.278,Z 658.656,A -85,B 0,C 180,E1 -9785.066,E2 -9785.066} C_VEL
LIN {X 0,Y 428.357,Z 672.341,A -85,B 0,C 180,E1 -9787.417,E2 -9787.417} C_VEL
LIN {X 0,Y 433.199,Z 700.361,A -85,B 0,C 180,E1 -9788.16,E2 -9788.16} C_VEL
LIN {X 0,Y 431.862,Z 805.846,A -85,B 0,C 180,E1 -9789.923,E2 -9789.923} C_VEL
LIN {X 0,Y 431.44,Z 819.969,A -85,B 0,C 180,E1 -9790.275,E2 -9790.275} C_VEL
LIN {X 0,Y 430.713,Z 834.425,A -85,B 0,C 180,E1 -9790.829,E2 -9790.829} C_VEL
LIN {X 0,Y 429.997,Z 847.411,A -85,B 0,C 180,E1 -9791.518,E2 -9791.518} C_VEL
LIN {X 0,Y 429.123,Z 859.839,A -85,B 0,C 180,E1 -9792.363,E2 -9792.363} C_VEL
LIN {X 0,Y 428.179,Z 872.394,A -85,B 0,C 180,E1 -9793.43,E2 -9793.43} C_VEL
LIN {X 0,Y 427.243,Z 883.739,A -85,B 0,C 180,E1 -9794.618,E2 -9794.618} C_VEL
LIN {X 0,Y 426.371,Z 894.03,A -85,B 0,C 180,E1 -9795.929,E2 -9795.929} C_VEL
LIN {X 0,Y 425.742,Z 903.651,A -85,B 0,C 180,E1 -9797.419,E2 -9797.419} C_VEL
LIN {X 0,Y 425.076,Z 912.239,A -85,B 0,C 180,E1 -9799.039,E2 -9799.039} C_VEL
LIN {X 0,Y 424.696,Z 918.512,A -85,B 0,C 180,E1 -9800.475,E2 -9800.475} C_VEL
LIN {X 0,Y 424.337,Z 925.16,A -85,B 0,C 180,E1 -9802.386,E2 -9802.386} C_VEL
LIN {X 0,Y 424.203,Z 930.144,A -85,B 0,C 180,E1 -9804.295,E2 -9804.295} C_VEL
LIN {X 0,Y 424.093,Z 933.614,A -85,B 0,C 180,E1 -9806.199,E2 -9806.199} C_VEL
LIN {X 0,Y 424.137,Z 935.681,A -85,B 0,C 180,E1 -9808.101,E2 -9808.101} C_VEL
LIN {X 0,Y 424.106,Z 936.388,A -85,B 0,C 180,E1 -9810,E2 -9810} C_VEL
LIN {X 0,Y 424.136,Z 935.754,A -85,B 0,C 180,E1 -9811.899,E2 -9811.899} C_VEL
LIN {X 0,Y 424.092,Z 933.761,A -85,B 0,C 180,E1 -9813.801,E2 -9813.801} C_VEL
LIN {X 0,Y 424.202,Z 930.37,A -85,B 0,C 180,E1 -9815.705,E2 -9815.705} C_VEL
LIN {X 0,Y 424.317,Z 926.865,A -85,B 0,C 180,E1 -9817.136,E2 -9817.136} C_VEL
LIN {X 0,Y 424.496,Z 922.438,A -85,B 0,C 180,E1 -9818.569,E2 -9818.569} C_VEL
LIN {X 0,Y 424.841,Z 916.043,A -85,B 0,C 180,E1 -9820.244,E2 -9820.244} C_VEL
LIN {X 0,Y 425.495,Z 908.108,A -85,B 0,C 180,E1 -9821.915,E2 -9821.915} C_VEL
LIN {X 0,Y 426.124,Z 899.827,A -85,B 0,C 180,E1 -9823.35,E2 -9823.35} C_VEL
LIN {X 0,Y 426.918,Z 889.873,A -85,B 0,C 180,E1 -9824.783,E2 -9824.783} C_VEL
LIN {X 0,Y 427.841,Z 878.825,A -85,B 0,C 180,E1 -9826.093,E2 -9826.093} C_VEL
LIN {X 0,Y 428.974,Z 866.519,A -85,B 0,C 180,E1 -9827.274,E2 -9827.274} C_VEL
LIN {X 0,Y 429.889,Z 854.35,A -85,B 0,C 180,E1 -9828.219,E2 -9828.219} C_VEL
LIN {X 0,Y 430.795,Z 840.849,A -85,B 0,C 180,E1 -9829.043,E2 -9829.043} C_VEL
LIN {X 0,Y 431.628,Z 826.737,A -85,B 0,C 180,E1 -9829.685,E2 -9829.685} C_VEL
LIN {X 0,Y 432.236,Z 812.922,A -85,B 0,C 180,E1 -9830.12,E2 -9830.12} C_VEL
LIN {X 0,Y 432.648,Z 790.799,A -85,B 0,C 180,E1 -9830.534,E2 -9830.534} C_VEL
LIN {X 0,Y 433.851,Z 700.687,A -85,B 0,C 180,E1 -9832.054,E2 -9832.054} C_VEL
LIN {X 0,Y 429.187,Z 674.894,A -85,B 0,C 180,E1 -9832.785,E2 -9832.785} C_VEL
LIN {X 0,Y 428.69,Z 672.121,A -85,B 0,C 180,E1 -9832.889,E2 -9832.889} C_VEL
LIN {X 0,Y 430.099,Z 654.3,A -85,B 0,C 180,E1 -9836.009,E2 -9836.009} C_VEL
LIN {X 0,Y 429.391,Z 649.047,A -85,B 0,C 180,E1 -9837.013,E2 -9837.013} C_VEL
LIN {X 0,Y 426.04,Z 634.675,A -85,B 0,C 180,E1 -9839.934,E2 -9839.934} C_VEL
LIN {X 0,Y 425.313,Z 631.631,A -85,B 0,C 180,E1 -9840.606,E2 -9840.606} C_VEL
LIN {X 0,Y 425.312,Z 631.626,A -85,B 0,C 180,E1 -9844.288,E2 -9844.288} C_VEL
LIN {X 0,Y 425.287,Z 631.634,A -85,B 0,C 180,E1 -9847.693,E2 -9847.693} C_VEL
LIN {X 0,Y 425.297,Z 631.626,A -85,B 0,C 180,E1 -9850.523,E2 -9850.523} C_VEL
LIN {X 0,Y 425.264,Z 631.633,A -85,B 0,C 180,E1 -9853.352,E2 -9853.352} C_VEL
LIN {X 0,Y 425.258,Z 631.634,A -85,B 0,C 180,E1 -9856.649,E2 -9856.649} C_VEL
LIN {X 0,Y 425.3,Z 631.631,A -85,B 0,C 180,E1 -9859.477,E2 -9859.477} C_VEL
LIN {X 0,Y 425.287,Z 631.619,A -85,B 0,C 180,E1 -9862.487,E2 -9862.487} C_VEL
LIN {X 0,Y 425.309,Z 631.632,A -85,B 0,C 180,E1 -9865.818,E2 -9865.818} C_VEL
LIN {X 0,Y 425.291,Z 631.615,A -85,B 0,C 180,E1 -9869.239,E2 -9869.239} C_VEL
LIN {X 0,Y 425.351,Z 631.622,A -85,B 0,C 180,E1 -9872.443,E2 -9872.443} C_VEL
LIN {X 0,Y 425.352,Z 631.625,A -85,B 0,C 180,E1 -9875.602,E2 -9875.602} C_VEL
LIN {X 0,Y 425.295,Z 631.629,A -85,B 0,C 180,E1 -9878.682,E2 -9878.682} C_VEL
LIN {X 0,Y 425.335,Z 631.625,A -85,B 0,C 180,E1 -9881.703,E2 -9881.703} C_VEL
LIN {X 0,Y 425.358,Z 631.622,A -85,B 0,C 180,E1 -9884.671,E2 -9884.671} C_VEL
LIN {X 0,Y 425.413,Z 631.614,A -85,B 0,C 180,E1 -9887.598,E2 -9887.598} C_VEL
LIN {X 0,Y 425.444,Z 631.606,A -85,B 0,C 180,E1 -9891.45,E2 -9891.45} C_VEL
LIN {X 0,Y 425.553,Z 631.6,A -85,B 0,C 180,E1 -9894.313,E2 -9894.313} C_VEL
LIN {X 0,Y 425.574,Z 631.599,A -85,B 0,C 180,E1 -9898.108,E2 -9898.108} C_VEL
LIN {X 0,Y 425.703,Z 631.581,A -85,B 0,C 180,E1 -9900,E2 -9900} C_VEL
LIN {X 0,Y 425.547,Z 631.601,A -85,B 0,C 180,E1 -9902.84,E2 -9902.84} C_VEL
LIN {X 0,Y 425.525,Z 631.604,A -85,B 0,C 180,E1 -9906.639,E2 -9906.639} C_VEL
LIN {X 0,Y 425.402,Z 631.614,A -85,B 0,C 180,E1 -9909.51,E2 -9909.51} C_VEL
LIN {X 0,Y 425.395,Z 631.62,A -85,B 0,C 180,E1 -9912.904,E2 -9912.904} C_VEL
LIN {X 0,Y 425.363,Z 631.625,A -85,B 0,C 180,E1 -9916.605,E2 -9916.605} C_VEL
LIN {X 0,Y 425.33,Z 631.621,A -85,B 0,C 180,E1 -9919.636,E2 -9919.636} C_VEL
LIN {X 0,Y 425.29,Z 631.634,A -85,B 0,C 180,E1 -9922.339,E2 -9922.339} C_VEL
LIN {X 0,Y 425.324,Z 631.628,A -85,B 0,C 180,E1 -9924.658,E2 -9924.658} C_VEL
LIN {X 0,Y 425.274,Z 631.625,A -85,B 0,C 180,E1 -9927.563,E2 -9927.563} C_VEL
LIN {X 0,Y 425.292,Z 631.625,A -85,B 0,C 180,E1 -9930.761,E2 -9930.761} C_VEL
LIN {X 0,Y 425.312,Z 631.625,A -85,B 0,C 180,E1 -9934.288,E2 -9934.288} C_VEL
LIN {X 0,Y 425.279,Z 631.634,A -85,B 0,C 180,E1 -9937.695,E2 -9937.695} C_VEL
LIN {X 0,Y 425.256,Z 631.63,A -85,B 0,C 180,E1 -9940.516,E2 -9940.516} C_VEL
LIN {X 0,Y 425.26,Z 631.636,A -85,B 0,C 180,E1 -9943.957,E2 -9943.957} C_VEL
LIN {X 0,Y 425.249,Z 631.638,A -85,B 0,C 180,E1 -9946.651,E2 -9946.651} C_VEL
LIN {X 0,Y 425.263,Z 631.639,A -85,B 0,C 180,E1 -9949.87,E2 -9949.87} C_VEL
LIN {X 0,Y 425.279,Z 631.635,A -85,B 0,C 180,E1 -9952.489,E2 -9952.489} C_VEL
LIN {X 0,Y 425.289,Z 631.633,A -85,B 0,C 180,E1 -9955.816,E2 -9955.816} C_VEL
LIN {X 0,Y 425.301,Z 631.675,A -85,B 0,C 180,E1 -9959.427,E2 -9959.427} C_VEL
LIN {X 0,Y 427.493,Z 641.855,A -85,B 0,C 180,E1 -9961.842,E2 -9961.842} C_VEL
LIN {X 0,Y 427.83,Z 643.27,A -85,B 0,C 180,E1 -9962.144,E2 -9962.144} C_VEL
LIN {X 0,Y 431.282,Z 652.64,A -85,B 0,C 180,E1 -9962.522,E2 -9962.522} C_VEL
LIN {X 0,Y 434.26,Z 666.129,A -85,B 0,C 180,E1 -9962.939,E2 -9962.939} C_VEL
LIN {X 0,Y 432.683,Z 778.828,A -85,B 0,C 180,E1 -9964.859,E2 -9964.859} C_VEL
LIN {X 0,Y 432.125,Z 793.357,A -85,B 0,C 180,E1 -9965.285,E2 -9965.285} C_VEL
LIN {X 0,Y 431.339,Z 807.455,A -85,B 0,C 180,E1 -9965.899,E2 -9965.899} C_VEL
LIN {X 0,Y 430.572,Z 820.688,A -85,B 0,C 180,E1 -9966.683,E2 -9966.683} C_VEL
LIN {X 0,Y 429.64,Z 833.439,A -85,B 0,C 180,E1 -9967.647,E2 -9967.647} C_VEL
LIN {X 0,Y 428.744,Z 845.012,A -85,B 0,C 180,E1 -9968.736,E2 -9968.736} C_VEL
LIN {X 0,Y 427.919,Z 854.611,A -85,B 0,C 180,E1 -9969.825,E2 -9969.825} C_VEL
LIN {X 0,Y 426.936,Z 865.252,A -85,B 0,C 180,E1 -9971.277,E2 -9971.277} C_VEL
LIN {X 0,Y 426.371,Z 871.569,A -85,B 0,C 180,E1 -9972.299,E2 -9972.299} C_VEL
LIN {X 0,Y 425.39,Z 875.194,A -85,B 0,C 180,E1 -9972.924,E2 -9972.924} C_VEL
LIN {X 0,Y 422.053,Z 880.737,A -85,B 0,C 180,E1 -9973.944,E2 -9973.944} C_VEL
LIN {X 0,Y 418.803,Z 885.786,A -85,B 0,C 180,E1 -9975.019,E2 -9975.019} C_VEL
LIN {X 0,Y 417.959,Z 888.478,A -85,B 0,C 180,E1 -9975.723,E2 -9975.723} C_VEL
LIN {X 0,Y 417.551,Z 894.033,A -85,B 0,C 180,E1 -9977.484,E2 -9977.484} C_VEL
LIN {X 0,Y 417.305,Z 898.432,A -85,B 0,C 180,E1 -9979.324,E2 -9979.324} C_VEL
LIN {X 0,Y 417.101,Z 901.667,A -85,B 0,C 180,E1 -9981.278,E2 -9981.278} C_VEL
LIN {X 0,Y 417.127,Z 903.493,A -85,B 0,C 180,E1 -9983.227,E2 -9983.227} C_VEL
LIN {X 0,Y 417.059,Z 903.997,A -85,B 0,C 180,E1 -9985.167,E2 -9985.167} C_VEL
LIN {X 0,Y 417.091,Z 903.187,A -85,B 0,C 180,E1 -9987.103,E2 -9987.103} C_VEL
LIN {X 0,Y 417.084,Z 901.061,A -85,B 0,C 180,E1 -9989.035,E2 -9989.035} C_VEL
LIN {X 0,Y 417.193,Z 897.565,A -85,B 0,C 180,E1 -9990.965,E2 -9990.965} C_VEL
LIN {X 0,Y 417.513,Z 892.594,A -85,B 0,C 180,E1 -9992.895,E2 -9992.895} C_VEL
LIN {X 0,Y 418.131,Z 885.987,A -85,B 0,C 180,E1 -9994.821,E2 -9994.821} C_VEL
LIN {X 0,Y 418.765,Z 878.63,A -85,B 0,C 180,E1 -9996.505,E2 -9996.505} C_VEL
LIN {X 0,Y 419.335,Z 870.1,A -85,B 0,C 180,E1 -9998.095,E2 -9998.095} C_VEL
LIN {X 0,Y 420.188,Z 861.18,A -85,B 0,C 180,E1 -9999.465,E2 -9999.465} C_VEL
LIN {X 0,Y 421.146,Z 850.496,A -85,B 0,C 180,E1 -10000.821,E2 -10000.821} C_VEL
LIN {X 0,Y 422.055,Z 839.048,A -85,B 0,C 180,E1 -10002.014,E2 -10002.014} C_VEL
LIN {X 0,Y 422.999,Z 826.342,A -85,B 0,C 180,E1 -10003.084,E2 -10003.084} C_VEL
LIN {X 0,Y 423.802,Z 813.933,A -85,B 0,C 180,E1 -10003.914,E2 -10003.914} C_VEL
LIN {X 0,Y 424.498,Z 800.127,A -85,B 0,C 180,E1 -10004.624,E2 -10004.624} C_VEL
LIN {X 0,Y 425.028,Z 785.519,A -85,B 0,C 180,E1 -10005.157,E2 -10005.157} C_VEL
LIN {X 0,Y 425.35,Z 770.881,A -85,B 0,C 180,E1 -10005.483,E2 -10005.483} C_VEL
LIN {X 0,Y 426.835,Z 666.095,A -85,B 0,C 180,E1 -10007.254,E2 -10007.254} C_VEL
LIN {X 0,Y 423.187,Z 650.736,A -85,B 0,C 180,E1 -10007.717,E2 -10007.717} C_VEL
LIN {X 0,Y 420.469,Z 643.154,A -85,B 0,C 180,E1 -10008.018,E2 -10008.018} C_VEL
LIN {X 0,Y 418.285,Z 632.512,A -85,B 0,C 180,E1 -10010.5,E2 -10010.5} C_VEL
LIN {X 0,Y 418.258,Z 632.51,A -85,B 0,C 180,E1 -10013.783,E2 -10013.783} C_VEL
LIN {X 0,Y 418.202,Z 632.52,A -85,B 0,C 180,E1 -10017.04,E2 -10017.04} C_VEL
LIN {X 0,Y 418.24,Z 632.513,A -85,B 0,C 180,E1 -10020.273,E2 -10020.273} C_VEL
LIN {X 0,Y 418.231,Z 632.511,A -85,B 0,C 180,E1 -10023.679,E2 -10023.679} C_VEL
LIN {X 0,Y 418.237,Z 632.513,A -85,B 0,C 180,E1 -10027.225,E2 -10027.225} C_VEL
LIN {X 0,Y 418.21,Z 632.509,A -85,B 0,C 180,E1 -10030.867,E2 -10030.867} C_VEL
LIN {X 0,Y 418.205,Z 632.511,A -85,B 0,C 180,E1 -10033.728,E2 -10033.728} C_VEL
LIN {X 0,Y 418.203,Z 632.514,A -85,B 0,C 180,E1 -10036.447,E2 -10036.447} C_VEL
LIN {X 0,Y 418.209,Z 632.519,A -85,B 0,C 180,E1 -10039.133,E2 -10039.133} C_VEL
LIN {X 0,Y 418.238,Z 632.495,A -85,B 0,C 180,E1 -10042.775,E2 -10042.775} C_VEL
LIN {X 0,Y 418.25,Z 632.507,A -85,B 0,C 180,E1 -10046.323,E2 -10046.323} C_VEL
LIN {X 0,Y 418.245,Z 632.504,A -85,B 0,C 180,E1 -10049.727,E2 -10049.727} C_VEL
LIN {X 0,Y 418.22,Z 632.515,A -85,B 0,C 180,E1 -10053.017,E2 -10053.017} C_VEL
LIN {X 0,Y 418.261,Z 632.498,A -85,B 0,C 180,E1 -10056.217,E2 -10056.217} C_VEL
LIN {X 0,Y 418.253,Z 632.513,A -85,B 0,C 180,E1 -10059.337,E2 -10059.337} C_VEL
LIN {X 0,Y 418.283,Z 632.491,A -85,B 0,C 180,E1 -10062.396,E2 -10062.396} C_VEL
LIN {X 0,Y 418.306,Z 632.504,A -85,B 0,C 180,E1 -10065.403,E2 -10065.403} C_VEL
LIN {X 0,Y 418.317,Z 632.493,A -85,B 0,C 180,E1 -10068.369,E2 -10068.369} C_VEL
LIN {X 0,Y 418.381,Z 632.488,A -85,B 0,C 180,E1 -10071.304,E2 -10071.304} C_VEL
LIN {X 0,Y 418.492,Z 632.477,A -85,B 0,C 180,E1 -10074.217,E2 -10074.217} C_VEL
LIN {X 0,Y 418.543,Z 632.474,A -85,B 0,C 180,E1 -10078.075,E2 -10078.075} C_VEL
LIN {X 0,Y 418.672,Z 632.455,A -85,B 0,C 180,E1 -10080,E2 -10080} C_VEL
LIN {X 0,Y 418.502,Z 632.475,A -85,B 0,C 180,E1 -10082.887,E2 -10082.887} C_VEL
LIN {X 0,Y 418.502,Z 632.477,A -85,B 0,C 180,E1 -10085.783,E2 -10085.783} C_VEL
LIN {X 0,Y 418.399,Z 632.489,A -85,B 0,C 180,E1 -10088.695,E2 -10088.695} C_VEL
LIN {X 0,Y 418.317,Z 632.497,A -85,B 0,C 180,E1 -10091.631,E2 -10091.631} C_VEL
LIN {X 0,Y 418.309,Z 632.497,A -85,B 0,C 180,E1 -10094.597,E2 -10094.597} C_VEL
LIN {X 0,Y 418.292,Z 632.503,A -85,B 0,C 180,E1 -10097.603,E2 -10097.603} C_VEL
LIN {X 0,Y 418.252,Z 632.507,A -85,B 0,C 180,E1 -10100.663,E2 -10100.663} C_VEL
LIN {X 0,Y 418.277,Z 632.503,A -85,B 0,C 180,E1 -10103.782,E2 -10103.782} C_VEL
LIN {X 0,Y 418.312,Z 632.496,A -85,B 0,C 180,E1 -10107.07,E2 -10107.07} C_VEL
LIN {X 0,Y 418.246,Z 632.512,A -85,B 0,C 180,E1 -10110.272,E2 -10110.272} C_VEL
LIN {X 0,Y 418.25,Z 632.508,A -85,B 0,C 180,E1 -10113.677,E2 -10113.677} C_VEL
LIN {X 0,Y 418.248,Z 632.508,A -85,B 0,C 180,E1 -10117.223,E2 -10117.223} C_VEL
LIN {X 0,Y 418.266,Z 632.504,A -85,B 0,C 180,E1 -10119.68,E2 -10119.68} C_VEL
LIN {X 0,Y 418.247,Z 632.511,A -85,B 0,C 180,E1 -10122.323,E2 -10122.323} C_VEL
LIN {X 0,Y 418.24,Z 632.509,A -85,B 0,C 180,E1 -10125.109,E2 -10125.109} C_VEL
LIN {X 0,Y 418.244,Z 632.507,A -85,B 0,C 180,E1 -10127.767,E2 -10127.767} C_VEL
LIN {X 0,Y 418.261,Z 632.512,A -85,B 0,C 180,E1 -10130.618,E2 -10130.618} C_VEL
LIN {X 0,Y 418.248,Z 632.51,A -85,B 0,C 180,E1 -10133.976,E2 -10133.976} C_VEL
LIN {X 0,Y 418.259,Z 632.512,A -85,B 0,C 180,E1 -10137.156,E2 -10137.156} C_VEL
LIN {X 0,Y 418.298,Z 632.562,A -85,B 0,C 180,E1 -10139.671,E2 -10139.671} C_VEL
LIN {X 0,Y 421.357,Z 646.059,A -85,B 0,C 180,E1 -10142.37,E2 -10142.37} C_VEL
LIN {X 0,Y 422.78,Z 653.776,A -85,B 0,C 180,E1 -10143.852,E2 -10143.852} C_VEL
LIN {X 0,Y 421.595,Z 671.357,A -85,B 0,C 180,E1 -10146.937,E2 -10146.937} C_VEL
LIN {X 0,Y 421.556,Z 672.521,A -85,B 0,C 180,E1 -10147.083,E2 -10147.083} C_VEL
LIN {X 0,Y 426.565,Z 701.775,A -85,B 0,C 180,E1 -10147.858,E2 -10147.858} C_VEL
LIN {X 0,Y 425.087,Z 807.376,A -85,B 0,C 180,E1 -10149.652,E2 -10149.652} C_VEL
LIN {X 0,Y 424.608,Z 821.718,A -85,B 0,C 180,E1 -10150.039,E2 -10150.039} C_VEL
LIN {X 0,Y 423.917,Z 834.941,A -85,B 0,C 180,E1 -10150.573,E2 -10150.573} C_VEL
LIN {X 0,Y 423.128,Z 848.228,A -85,B 0,C 180,E1 -10151.301,E2 -10151.301} C_VEL
LIN {X 0,Y 422.211,Z 860.846,A -85,B 0,C 180,E1 -10152.19,E2 -10152.19} C_VEL
LIN {X 0,Y 421.19,Z 873.118,A -85,B 0,C 180,E1 -10153.272,E2 -10153.272} C_VEL
LIN {X 0,Y 420.231,Z 884.266,A -85,B 0,C 180,E1 -10154.479,E2 -10154.479} C_VEL
LIN {X 0,Y 419.274,Z 895.245,A -85,B 0,C 180,E1 -10155.933,E2 -10155.933} C_VEL
LIN {X 0,Y 418.664,Z 904.319,A -85,B 0,C 180,E1 -10157.395,E2 -10157.395} C_VEL
LIN {X 0,Y 417.961,Z 912.991,A -85,B 0,C 180,E1 -10159.096,E2 -10159.096} C_VEL
LIN {X 0,Y 417.525,Z 919.987,A -85,B 0,C 180,E1 -10160.798,E2 -10160.798} C_VEL
LIN {X 0,Y 417.242,Z 926.26,A -85,B 0,C 180,E1 -10162.742,E2 -10162.742} C_VEL
LIN {X 0,Y 417.12,Z 929.825,A -85,B 0,C 180,E1 -10164.198,E2 -10164.198} C_VEL
LIN {X 0,Y 417.008,Z 933.31,A -85,B 0,C 180,E1 -10166.134,E2 -10166.134} C_VEL
LIN {X 0,Y 417.064,Z 935.392,A -85,B 0,C 180,E1 -10168.069,E2 -10168.069} C_VEL
LIN {X 0,Y 417.024,Z 936.113,A -85,B 0,C 180,E1 -10170,E2 -10170} C_VEL
LIN {X 0,Y 417.062,Z 935.494,A -85,B 0,C 180,E1 -10171.931,E2 -10171.931} C_VEL
LIN {X 0,Y 417.007,Z 933.518,A -85,B 0,C 180,E1 -10173.865,E2 -10173.865} C_VEL
LIN {X 0,Y 417.119,Z 930.141,A -85,B 0,C 180,E1 -10175.802,E2 -10175.802} C_VEL
LIN {X 0,Y 417.242,Z 926.645,A -85,B 0,C 180,E1 -10177.257,E2 -10177.257} C_VEL
LIN {X 0,Y 417.534,Z 920.59,A -85,B 0,C 180,E1 -10179.201,E2 -10179.201} C_VEL
LIN {X 0,Y 417.975,Z 913.794,A -85,B 0,C 180,E1 -10180.904,E2 -10180.904} C_VEL
LIN {X 0,Y 418.671,Z 905.365,A -85,B 0,C 180,E1 -10182.605,E2 -10182.605} C_VEL
LIN {X 0,Y 419.41,Z 896.597,A -85,B 0,C 180,E1 -10184.062,E2 -10184.062} C_VEL
LIN {X 0,Y 420.35,Z 885.993,A -85,B 0,C 180,E1 -10185.516,E2 -10185.516} C_VEL
LIN {X 0,Y 421.344,Z 875.313,A -85,B 0,C 180,E1 -10186.722,E2 -10186.722} C_VEL
LIN {X 0,Y 422.375,Z 863.678,A -85,B 0,C 180,E1 -10187.803,E2 -10187.803} C_VEL
LIN {X 0,Y 423.464,Z 850.664,A -85,B 0,C 180,E1 -10188.774,E2 -10188.774} C_VEL
LIN {X 0,Y 424.294,Z 837.65,A -85,B 0,C 180,E1 -10189.535,E2 -10189.535} C_VEL
LIN {X 0,Y 425.125,Z 824.046,A -85,B 0,C 180,E1 -10190.125,E2 -10190.125} C_VEL
LIN {X 0,Y 425.701,Z 810.169,A -85,B 0,C 180,E1 -10190.538,E2 -10190.538} C_VEL
LIN {X 0,Y 427.356,Z 701.697,A -85,B 0,C 180,E1 -10192.411,E2 -10192.411} C_VEL
LIN {X 0,Y 422.67,Z 675.98,A -85,B 0,C 180,E1 -10193.16,E2 -10193.16} C_VEL
LIN {X 0,Y 421.896,Z 671.806,A -85,B 0,C 180,E1 -10193.316,E2 -10193.316} C_VEL
LIN {X 0,Y 423.276,Z 655.157,A -85,B 0,C 180,E1 -10196.285,E2 -10196.285} C_VEL
LIN {X 0,Y 421.491,Z 646.082,A -85,B 0,C 180,E1 -10198.102,E2 -10198.102} C_VEL
LIN {X 0,Y 418.826,Z 634.792,A -85,B 0,C 180,E1 -10200.468,E2 -10200.468} C_VEL
LIN {X 0,Y 418.233,Z 632.512,A -85,B 0,C 180,E1 -10200.963,E2 -10200.963} C_VEL
LIN {X 0,Y 418.249,Z 632.506,A -85,B 0,C 180,E1 -10203.677,E2 -10203.677} C_VEL
LIN {X 0,Y 418.247,Z 632.511,A -85,B 0,C 180,E1 -10207.223,E2 -10207.223} C_VEL
LIN {X 0,Y 418.262,Z 632.506,A -85,B 0,C 180,E1 -10209.681,E2 -10209.681} C_VEL
LIN {X 0,Y 418.248,Z 632.509,A -85,B 0,C 180,E1 -10212.324,E2 -10212.324} C_VEL
LIN {X 0,Y 418.238,Z 632.509,A -85,B 0,C 180,E1 -10215.109,E2 -10215.109} C_VEL
LIN {X 0,Y 418.257,Z 632.501,A -85,B 0,C 180,E1 -10217.769,E2 -10217.769} C_VEL
LIN {X 0,Y 418.269,Z 632.506,A -85,B 0,C 180,E1 -10220.617,E2 -10220.617} C_VEL
LIN {X 0,Y 418.247,Z 632.508,A -85,B 0,C 180,E1 -10223.976,E2 -10223.976} C_VEL
LIN {X 0,Y 418.258,Z 632.505,A -85,B 0,C 180,E1 -10227.156,E2 -10227.156} C_VEL
LIN {X 0,Y 418.269,Z 632.502,A -85,B 0,C 180,E1 -10230.896,E2 -10230.896} C_VEL
LIN {X 0,Y 418.272,Z 632.506,A -85,B 0,C 180,E1 -10234.096,E2 -10234.096} C_VEL
LIN {X 0,Y 418.239,Z 632.506,A -85,B 0,C 180,E1 -10237.264,E2 -10237.264} C_VEL
LIN {X 0,Y 418.285,Z 632.503,A -85,B 0,C 180,E1 -10240.364,E2 -10240.364} C_VEL
LIN {X 0,Y 418.327,Z 632.498,A -85,B 0,C 180,E1 -10243.405,E2 -10243.405} C_VEL
LIN {X 0,Y 418.347,Z 632.493,A -85,B 0,C 180,E1 -10246.999,E2 -10246.999} C_VEL
LIN {X 0,Y 418.343,Z 632.494,A -85,B 0,C 180,E1 -10250.329,E2 -10250.329} C_VEL
LIN {X 0,Y 418.49,Z 632.478,A -85,B 0,C 180,E1 -10253.249,E2 -10253.249} C_VEL
LIN {X 0,Y 418.34,Z 632.491,A -85,B 0,C 180,E1 -10255.182,E2 -10255.182} C_VEL
LIN {X 0,Y 418.543,Z 632.475,A -85,B 0,C 180,E1 -10258.076,E2 -10258.076} C_VEL
LIN {X 0,Y 418.673,Z 632.456,A -85,B 0,C 180,E1 -10260,E2 -10260} C_VEL
LIN {X 0,Y 418.503,Z 632.478,A -85,B 0,C 180,E1 -10262.888,E2 -10262.888} C_VEL
LIN {X 0,Y 418.489,Z 632.482,A -85,B 0,C 180,E1 -10266.751,E2 -10266.751} C_VEL
LIN {X 0,Y 418.342,Z 632.493,A -85,B 0,C 180,E1 -10269.672,E2 -10269.672} C_VEL
LIN {X 0,Y 418.348,Z 632.497,A -85,B 0,C 180,E1 -10273.001,E2 -10273.001} C_VEL
LIN {X 0,Y 418.314,Z 632.505,A -85,B 0,C 180,E1 -10276.736,E2 -10276.736} C_VEL
LIN {X 0,Y 418.273,Z 632.5,A -85,B 0,C 180,E1 -10279.79,E2 -10279.79} C_VEL
LIN {X 0,Y 418.234,Z 632.512,A -85,B 0,C 180,E1 -10282.737,E2 -10282.737} C_VEL
LIN {X 0,Y 418.24,Z 632.509,A -85,B 0,C 180,E1 -10285.906,E2 -10285.906} C_VEL
LIN {X 0,Y 418.263,Z 632.492,A -85,B 0,C 180,E1 -10289.163,E2 -10289.163} C_VEL
LIN {X 0,Y 418.259,Z 632.513,A -85,B 0,C 180,E1 -10292.844,E2 -10292.844} C_VEL
LIN {X 0,Y 418.247,Z 632.509,A -85,B 0,C 180,E1 -10296.238,E2 -10296.238} C_VEL
LIN {X 0,Y 418.212,Z 632.508,A -85,B 0,C 180,E1 -10299.687,E2 -10299.687} C_VEL
LIN {X 0,Y 418.214,Z 632.512,A -85,B 0,C 180,E1 -10302.319,E2 -10302.319} C_VEL
LIN {X 0,Y 418.238,Z 632.508,A -85,B 0,C 180,E1 -10305.109,E2 -10305.109} C_VEL
LIN {X 0,Y 418.222,Z 632.516,A -85,B 0,C 180,E1 -10307.765,E2 -10307.765} C_VEL
LIN {X 0,Y 418.243,Z 632.515,A -85,B 0,C 180,E1 -10311.557,E2 -10311.557} C_VEL
LIN {X 0,Y 418.254,Z 632.51,A -85,B 0,C 180,E1 -10315.158,E2 -10315.158} C_VEL
LIN {X 0,Y 418.246,Z 632.499,A -85,B 0,C 180,E1 -10317.472,E2 -10317.472} C_VEL
LIN {X 0,Y 418.243,Z 632.579,A -85,B 0,C 180,E1 -10319.071,E2 -10319.071} C_VEL
LIN {X 0,Y 420.607,Z 643.329,A -85,B 0,C 180,E1 -10321.672,E2 -10321.672} C_VEL
LIN {X 0,Y 425,Z 654.701,A -85,B 0,C 180,E1 -10322.176,E2 -10322.176} C_VEL
LIN {X 0,Y 427.738,Z 667.36,A -85,B 0,C 180,E1 -10322.574,E2 -10322.574} C_VEL
